			//Type Arrays
			//ARRAY OF BOOL
			IF FIND(Lynus_Standards.GVL_Communicator.arrInterfaceInfoAlVariables[byReadWriteArrayNumber,udiActiveNumberOfSymbol_ReadAds].sSymbolType,'OF BOOL') <> 0 THEN
				stADSRead_ReadAds[udiActiveNumberOfSymbol_ReadAds].sFullSymbolName := Lynus_Standards.GVL_Communicator.arrInterfaceInfoAlVariables[byReadWriteArrayNumber,udiActiveNumberOfSymbol_ReadAds].sFullSymbolName;
					stADSRead_ReadAds[udiActiveNumberOfSymbol_ReadAds].arrValue := arrValueDefault_ReadAds;	
						IF Lynus_Standards.GVL_Communicator.arrInterfaceInfoAlVariables[byReadWriteArrayNumber,udiActiveNumberOfSymbol_ReadAds].uiSizeArray <= Lynus_Standards.Constants_Communicator.bySizeOfValueArray THEN  
							FOR uiLPWriteValueByArray_ReadAds := 1 TO Lynus_Standards.GVL_Communicator.arrInterfaceInfoAlVariables[byReadWriteArrayNumber,udiActiveNumberOfSymbol_ReadAds].uiSizeArray BY 1 DO 	
								stADSRead_ReadAds[udiActiveNumberOfSymbol_ReadAds].arrValue[uiLPWriteValueByArray_ReadAds] := BYTE_TO_STRING(arrValueAfterRead_ReadAds[uiLPWriteValueByArray_ReadAds]);
							END_FOR 
						END_IF
			END_IF 
				//ARRAY OF BYTE
				IF FIND(Lynus_Standards.GVL_Communicator.arrInterfaceInfoAlVariables[byReadWriteArrayNumber,udiActiveNumberOfSymbol_ReadAds].sSymbolType,'OF BYTE') <> 0 THEN
					stADSRead_ReadAds[udiActiveNumberOfSymbol_ReadAds].sFullSymbolName := Lynus_Standards.GVL_Communicator.arrInterfaceInfoAlVariables[byReadWriteArrayNumber,udiActiveNumberOfSymbol_ReadAds].sFullSymbolName;
						stADSRead_ReadAds[udiActiveNumberOfSymbol_ReadAds].arrValue := arrValueDefault_ReadAds;	
							IF Lynus_Standards.GVL_Communicator.arrInterfaceInfoAlVariables[byReadWriteArrayNumber,udiActiveNumberOfSymbol_ReadAds].uiSizeArray <= Lynus_Standards.Constants_Communicator.bySizeOfValueArray THEN  
								FOR uiLPWriteValueByArray_ReadAds := 1 TO Lynus_Standards.GVL_Communicator.arrInterfaceInfoAlVariables[byReadWriteArrayNumber,udiActiveNumberOfSymbol_ReadAds].uiSizeArray BY 1 DO 	
									stADSRead_ReadAds[udiActiveNumberOfSymbol_ReadAds].arrValue[uiLPWriteValueByArray_ReadAds] := BYTE_TO_STRING(arrValueAfterRead_ReadAds[uiLPWriteValueByArray_ReadAds]);
								END_FOR 
							END_IF
				END_IF
			//ARRAY OF WORD
			IF FIND(Lynus_Standards.GVL_Communicator.arrInterfaceInfoAlVariables[byReadWriteArrayNumber,udiActiveNumberOfSymbol_ReadAds].sSymbolType,'OF WORD') <> 0 THEN
				stADSRead_ReadAds[udiActiveNumberOfSymbol_ReadAds].sFullSymbolName := Lynus_Standards.GVL_Communicator.arrInterfaceInfoAlVariables[byReadWriteArrayNumber,udiActiveNumberOfSymbol_ReadAds].sFullSymbolName;
					stADSRead_ReadAds[udiActiveNumberOfSymbol_ReadAds].arrValue := arrValueDefault_ReadAds;	
						IF Lynus_Standards.GVL_Communicator.arrInterfaceInfoAlVariables[byReadWriteArrayNumber,udiActiveNumberOfSymbol_ReadAds].uiSizeArray <= Lynus_Standards.Constants_Communicator.bySizeOfValueArray THEN  
							FOR uiLPWriteValueByArray_ReadAds := 1 TO Lynus_Standards.GVL_Communicator.arrInterfaceInfoAlVariables[byReadWriteArrayNumber,udiActiveNumberOfSymbol_ReadAds].uiSizeArray BY 1 DO
								arrCounterWriteValueInArray_ReadAds[1] := LIMIT(1,arrCounterWriteValueInArray_ReadAds[1],1600); arrCounterWriteValueInArray_ReadAds[2] := LIMIT(2,arrCounterWriteValueInArray_ReadAds[2],1600);
									stADSRead_ReadAds[udiActiveNumberOfSymbol_ReadAds].arrValue[uiLPWriteValueByArray_ReadAds] := WORD_TO_STRING(SHL(BYTE_TO_WORD(arrValueAfterRead_ReadAds[arrCounterWriteValueInArray_ReadAds[2]]),8) + BYTE_TO_WORD(arrValueAfterRead_ReadAds[arrCounterWriteValueInArray_ReadAds[1]]));;
								arrCounterWriteValueInArray_ReadAds[1] := arrCounterWriteValueInArray_ReadAds[1] + 2; arrCounterWriteValueInArray_ReadAds[2] := arrCounterWriteValueInArray_ReadAds[2] + 2;
							END_FOR 
						END_IF
			END_IF
				//ARRAY OF DWORD	
				IF FIND(Lynus_Standards.GVL_Communicator.arrInterfaceInfoAlVariables[byReadWriteArrayNumber,udiActiveNumberOfSymbol_ReadAds].sSymbolType,'OF DWORD') <> 0 THEN
					stADSRead_ReadAds[udiActiveNumberOfSymbol_ReadAds].sFullSymbolName := Lynus_Standards.GVL_Communicator.arrInterfaceInfoAlVariables[byReadWriteArrayNumber,udiActiveNumberOfSymbol_ReadAds].sFullSymbolName;
						stADSRead_ReadAds[udiActiveNumberOfSymbol_ReadAds].arrValue := arrValueDefault_ReadAds;	
							IF Lynus_Standards.GVL_Communicator.arrInterfaceInfoAlVariables[byReadWriteArrayNumber,udiActiveNumberOfSymbol_ReadAds].uiSizeArray <= Lynus_Standards.Constants_Communicator.bySizeOfValueArray THEN  
								FOR uiLPWriteValueByArray_ReadAds := 1 TO Lynus_Standards.GVL_Communicator.arrInterfaceInfoAlVariables[byReadWriteArrayNumber,udiActiveNumberOfSymbol_ReadAds].uiSizeArray BY 1 DO
									arrCounterWriteValueInArray_ReadAds[1] := LIMIT(1,arrCounterWriteValueInArray_ReadAds[1],1600); arrCounterWriteValueInArray_ReadAds[2] := LIMIT(2,arrCounterWriteValueInArray_ReadAds[2],1600);
										arrCounterWriteValueInArray_ReadAds[3] := LIMIT(3,arrCounterWriteValueInArray_ReadAds[3],1600); arrCounterWriteValueInArray_ReadAds[4] := LIMIT(4,arrCounterWriteValueInArray_ReadAds[4],1600);
											stADSRead_ReadAds[udiActiveNumberOfSymbol_ReadAds].arrValue[uiLPWriteValueByArray_ReadAds] := DWORD_TO_STRING(SHL(BYTE_TO_DWORD(arrValueAfterRead_ReadAds[arrCounterWriteValueInArray_ReadAds[4]]),24) + SHL(BYTE_TO_DWORD(arrValueAfterRead_ReadAds[arrCounterWriteValueInArray_ReadAds[3]]),16) + SHL(BYTE_TO_DWORD(arrValueAfterRead_ReadAds[arrCounterWriteValueInArray_ReadAds[2]]),8) + BYTE_TO_DWORD(arrValueAfterRead_ReadAds[arrCounterWriteValueInArray_ReadAds[1]]));
									arrCounterWriteValueInArray_ReadAds[1] := arrCounterWriteValueInArray_ReadAds[1] + 4; arrCounterWriteValueInArray_ReadAds[2] := arrCounterWriteValueInArray_ReadAds[2] + 4;
										arrCounterWriteValueInArray_ReadAds[3] := arrCounterWriteValueInArray_ReadAds[3] + 4; arrCounterWriteValueInArray_ReadAds[4] := arrCounterWriteValueInArray_ReadAds[4] + 4;
								END_FOR 
							END_IF
				END_IF
			//ARRAY OF SINT
			IF FIND(Lynus_Standards.GVL_Communicator.arrInterfaceInfoAlVariables[byReadWriteArrayNumber,udiActiveNumberOfSymbol_ReadAds].sSymbolType,'OF SINT') <> 0 THEN
				stADSRead_ReadAds[udiActiveNumberOfSymbol_ReadAds].sFullSymbolName := Lynus_Standards.GVL_Communicator.arrInterfaceInfoAlVariables[byReadWriteArrayNumber,udiActiveNumberOfSymbol_ReadAds].sFullSymbolName;
					stADSRead_ReadAds[udiActiveNumberOfSymbol_ReadAds].arrValue := arrValueDefault_ReadAds;	
						IF Lynus_Standards.GVL_Communicator.arrInterfaceInfoAlVariables[byReadWriteArrayNumber,udiActiveNumberOfSymbol_ReadAds].uiSizeArray <= Lynus_Standards.Constants_Communicator.bySizeOfValueArray THEN  
							FOR uiLPWriteValueByArray_ReadAds := 1 TO Lynus_Standards.GVL_Communicator.arrInterfaceInfoAlVariables[byReadWriteArrayNumber,udiActiveNumberOfSymbol_ReadAds].uiSizeArray BY 1 DO 	
								stADSRead_ReadAds[udiActiveNumberOfSymbol_ReadAds].arrValue[uiLPWriteValueByArray_ReadAds] := SINT_TO_STRING(BYTE_TO_SINT(arrValueAfterRead_ReadAds[uiLPWriteValueByArray_ReadAds]));
							END_FOR 
						END_IF
			END_IF
				//ARRAY OF USINT
				IF FIND(Lynus_Standards.GVL_Communicator.arrInterfaceInfoAlVariables[byReadWriteArrayNumber,udiActiveNumberOfSymbol_ReadAds].sSymbolType,'OF USINT') <> 0 THEN
					stADSRead_ReadAds[udiActiveNumberOfSymbol_ReadAds].sFullSymbolName := Lynus_Standards.GVL_Communicator.arrInterfaceInfoAlVariables[byReadWriteArrayNumber,udiActiveNumberOfSymbol_ReadAds].sFullSymbolName;
						stADSRead_ReadAds[udiActiveNumberOfSymbol_ReadAds].arrValue := arrValueDefault_ReadAds;	
							IF Lynus_Standards.GVL_Communicator.arrInterfaceInfoAlVariables[byReadWriteArrayNumber,udiActiveNumberOfSymbol_ReadAds].uiSizeArray <= Lynus_Standards.Constants_Communicator.bySizeOfValueArray THEN  
								FOR uiLPWriteValueByArray_ReadAds := 1 TO Lynus_Standards.GVL_Communicator.arrInterfaceInfoAlVariables[byReadWriteArrayNumber,udiActiveNumberOfSymbol_ReadAds].uiSizeArray BY 1 DO 	
									stADSRead_ReadAds[udiActiveNumberOfSymbol_ReadAds].arrValue[uiLPWriteValueByArray_ReadAds] := USINT_TO_STRING(BYTE_TO_USINT(arrValueAfterRead_ReadAds[uiLPWriteValueByArray_ReadAds]));
								END_FOR 
							END_IF
				END_IF
			//ARRAY OF INT
			IF FIND(Lynus_Standards.GVL_Communicator.arrInterfaceInfoAlVariables[byReadWriteArrayNumber,udiActiveNumberOfSymbol_ReadAds].sSymbolType,'OF INT') <> 0 THEN
				stADSRead_ReadAds[udiActiveNumberOfSymbol_ReadAds].sFullSymbolName := Lynus_Standards.GVL_Communicator.arrInterfaceInfoAlVariables[byReadWriteArrayNumber,udiActiveNumberOfSymbol_ReadAds].sFullSymbolName;
					stADSRead_ReadAds[udiActiveNumberOfSymbol_ReadAds].arrValue := arrValueDefault_ReadAds;	
						IF Lynus_Standards.GVL_Communicator.arrInterfaceInfoAlVariables[byReadWriteArrayNumber,udiActiveNumberOfSymbol_ReadAds].uiSizeArray <= Lynus_Standards.Constants_Communicator.bySizeOfValueArray THEN  
							FOR uiLPWriteValueByArray_ReadAds := 1 TO Lynus_Standards.GVL_Communicator.arrInterfaceInfoAlVariables[byReadWriteArrayNumber,udiActiveNumberOfSymbol_ReadAds].uiSizeArray BY 1 DO
								arrCounterWriteValueInArray_ReadAds[1] := LIMIT(1,arrCounterWriteValueInArray_ReadAds[1],1600); arrCounterWriteValueInArray_ReadAds[2] := LIMIT(2,arrCounterWriteValueInArray_ReadAds[2],1600);
									stADSRead_ReadAds[udiActiveNumberOfSymbol_ReadAds].arrValue[uiLPWriteValueByArray_ReadAds] := INT_TO_STRING(SHL(BYTE_TO_INT(arrValueAfterRead_ReadAds[arrCounterWriteValueInArray_ReadAds[2]]),8) + BYTE_TO_INT(arrValueAfterRead_ReadAds[arrCounterWriteValueInArray_ReadAds[1]]));;
								arrCounterWriteValueInArray_ReadAds[1] := arrCounterWriteValueInArray_ReadAds[1] + 2; arrCounterWriteValueInArray_ReadAds[2] := arrCounterWriteValueInArray_ReadAds[2] + 2;
							END_FOR 
						END_IF
			END_IF
				//ARRAY OF UINT
				IF FIND(Lynus_Standards.GVL_Communicator.arrInterfaceInfoAlVariables[byReadWriteArrayNumber,udiActiveNumberOfSymbol_ReadAds].sSymbolType,'OF UINT') <> 0 THEN
					stADSRead_ReadAds[udiActiveNumberOfSymbol_ReadAds].sFullSymbolName := Lynus_Standards.GVL_Communicator.arrInterfaceInfoAlVariables[byReadWriteArrayNumber,udiActiveNumberOfSymbol_ReadAds].sFullSymbolName;
						stADSRead_ReadAds[udiActiveNumberOfSymbol_ReadAds].arrValue := arrValueDefault_ReadAds;	
							IF Lynus_Standards.GVL_Communicator.arrInterfaceInfoAlVariables[byReadWriteArrayNumber,udiActiveNumberOfSymbol_ReadAds].uiSizeArray <= Lynus_Standards.Constants_Communicator.bySizeOfValueArray THEN  
								FOR uiLPWriteValueByArray_ReadAds := 1 TO Lynus_Standards.GVL_Communicator.arrInterfaceInfoAlVariables[byReadWriteArrayNumber,udiActiveNumberOfSymbol_ReadAds].uiSizeArray BY 1 DO
									arrCounterWriteValueInArray_ReadAds[1] := LIMIT(1,arrCounterWriteValueInArray_ReadAds[1],1600); arrCounterWriteValueInArray_ReadAds[2] := LIMIT(2,arrCounterWriteValueInArray_ReadAds[2],1600);
										stADSRead_ReadAds[udiActiveNumberOfSymbol_ReadAds].arrValue[uiLPWriteValueByArray_ReadAds] := UINT_TO_STRING(SHL(BYTE_TO_UINT(arrValueAfterRead_ReadAds[arrCounterWriteValueInArray_ReadAds[2]]),8) + BYTE_TO_UINT(arrValueAfterRead_ReadAds[arrCounterWriteValueInArray_ReadAds[1]]));;
									arrCounterWriteValueInArray_ReadAds[1] := arrCounterWriteValueInArray_ReadAds[1] + 2; arrCounterWriteValueInArray_ReadAds[2] := arrCounterWriteValueInArray_ReadAds[2] + 2;
								END_FOR 
							END_IF
				END_IF
			//ARRAY OF DINT	
			IF FIND(Lynus_Standards.GVL_Communicator.arrInterfaceInfoAlVariables[byReadWriteArrayNumber,udiActiveNumberOfSymbol_ReadAds].sSymbolType,'OF DINT') <> 0 THEN
				stADSRead_ReadAds[udiActiveNumberOfSymbol_ReadAds].sFullSymbolName := Lynus_Standards.GVL_Communicator.arrInterfaceInfoAlVariables[byReadWriteArrayNumber,udiActiveNumberOfSymbol_ReadAds].sFullSymbolName;
					stADSRead_ReadAds[udiActiveNumberOfSymbol_ReadAds].arrValue := arrValueDefault_ReadAds;	
						IF Lynus_Standards.GVL_Communicator.arrInterfaceInfoAlVariables[byReadWriteArrayNumber,udiActiveNumberOfSymbol_ReadAds].uiSizeArray <= Lynus_Standards.Constants_Communicator.bySizeOfValueArray THEN  
							FOR uiLPWriteValueByArray_ReadAds := 1 TO Lynus_Standards.GVL_Communicator.arrInterfaceInfoAlVariables[byReadWriteArrayNumber,udiActiveNumberOfSymbol_ReadAds].uiSizeArray BY 1 DO
								arrCounterWriteValueInArray_ReadAds[1] := LIMIT(1,arrCounterWriteValueInArray_ReadAds[1],1600); arrCounterWriteValueInArray_ReadAds[2] := LIMIT(2,arrCounterWriteValueInArray_ReadAds[2],1600);
									arrCounterWriteValueInArray_ReadAds[3] := LIMIT(3,arrCounterWriteValueInArray_ReadAds[3],1600); arrCounterWriteValueInArray_ReadAds[4] := LIMIT(4,arrCounterWriteValueInArray_ReadAds[4],1600);
										stADSRead_ReadAds[udiActiveNumberOfSymbol_ReadAds].arrValue[uiLPWriteValueByArray_ReadAds] := DINT_TO_STRING(SHL(BYTE_TO_DINT(arrValueAfterRead_ReadAds[arrCounterWriteValueInArray_ReadAds[4]]),24) + SHL(BYTE_TO_DINT(arrValueAfterRead_ReadAds[arrCounterWriteValueInArray_ReadAds[3]]),16) + SHL(BYTE_TO_DINT(arrValueAfterRead_ReadAds[arrCounterWriteValueInArray_ReadAds[2]]),8) + BYTE_TO_DINT(arrValueAfterRead_ReadAds[arrCounterWriteValueInArray_ReadAds[1]]));
								arrCounterWriteValueInArray_ReadAds[1] := arrCounterWriteValueInArray_ReadAds[1] + 4; arrCounterWriteValueInArray_ReadAds[2] := arrCounterWriteValueInArray_ReadAds[2] + 4;
									arrCounterWriteValueInArray_ReadAds[3] := arrCounterWriteValueInArray_ReadAds[3] + 4; arrCounterWriteValueInArray_ReadAds[4] := arrCounterWriteValueInArray_ReadAds[4] + 4;
							END_FOR 
						END_IF
			END_IF
				//ARRAY OF UDINT	
				IF FIND(Lynus_Standards.GVL_Communicator.arrInterfaceInfoAlVariables[byReadWriteArrayNumber,udiActiveNumberOfSymbol_ReadAds].sSymbolType,'OF UDINT') <> 0 THEN
					stADSRead_ReadAds[udiActiveNumberOfSymbol_ReadAds].sFullSymbolName := Lynus_Standards.GVL_Communicator.arrInterfaceInfoAlVariables[byReadWriteArrayNumber,udiActiveNumberOfSymbol_ReadAds].sFullSymbolName;
						stADSRead_ReadAds[udiActiveNumberOfSymbol_ReadAds].arrValue := arrValueDefault_ReadAds;	
							IF Lynus_Standards.GVL_Communicator.arrInterfaceInfoAlVariables[byReadWriteArrayNumber,udiActiveNumberOfSymbol_ReadAds].uiSizeArray <= Lynus_Standards.Constants_Communicator.bySizeOfValueArray THEN  
								FOR uiLPWriteValueByArray_ReadAds := 1 TO Lynus_Standards.GVL_Communicator.arrInterfaceInfoAlVariables[byReadWriteArrayNumber,udiActiveNumberOfSymbol_ReadAds].uiSizeArray BY 1 DO
									arrCounterWriteValueInArray_ReadAds[1] := LIMIT(1,arrCounterWriteValueInArray_ReadAds[1],1600); arrCounterWriteValueInArray_ReadAds[2] := LIMIT(2,arrCounterWriteValueInArray_ReadAds[2],1600);
										arrCounterWriteValueInArray_ReadAds[3] := LIMIT(3,arrCounterWriteValueInArray_ReadAds[3],1600); arrCounterWriteValueInArray_ReadAds[4] := LIMIT(4,arrCounterWriteValueInArray_ReadAds[4],1600);
											stADSRead_ReadAds[udiActiveNumberOfSymbol_ReadAds].arrValue[uiLPWriteValueByArray_ReadAds] := UDINT_TO_STRING(SHL(BYTE_TO_UDINT(arrValueAfterRead_ReadAds[arrCounterWriteValueInArray_ReadAds[4]]),24) + SHL(BYTE_TO_UDINT(arrValueAfterRead_ReadAds[arrCounterWriteValueInArray_ReadAds[3]]),16) + SHL(BYTE_TO_UDINT(arrValueAfterRead_ReadAds[arrCounterWriteValueInArray_ReadAds[2]]),8) + BYTE_TO_UDINT(arrValueAfterRead_ReadAds[arrCounterWriteValueInArray_ReadAds[1]]));
									arrCounterWriteValueInArray_ReadAds[1] := arrCounterWriteValueInArray_ReadAds[1] + 4; arrCounterWriteValueInArray_ReadAds[2] := arrCounterWriteValueInArray_ReadAds[2] + 4;
										arrCounterWriteValueInArray_ReadAds[3] := arrCounterWriteValueInArray_ReadAds[3] + 4; arrCounterWriteValueInArray_ReadAds[4] := arrCounterWriteValueInArray_ReadAds[4] + 4;
								END_FOR 
							END_IF
				END_IF
					//ARRAY OF LINT	
					IF FIND(Lynus_Standards.GVL_Communicator.arrInterfaceInfoAlVariables[byReadWriteArrayNumber,udiActiveNumberOfSymbol_ReadAds].sSymbolType,'OF LINT') <> 0 THEN
						stADSRead_ReadAds[udiActiveNumberOfSymbol_ReadAds].sFullSymbolName := Lynus_Standards.GVL_Communicator.arrInterfaceInfoAlVariables[byReadWriteArrayNumber,udiActiveNumberOfSymbol_ReadAds].sFullSymbolName;
							stADSRead_ReadAds[udiActiveNumberOfSymbol_ReadAds].arrValue := arrValueDefault_ReadAds;	
								IF Lynus_Standards.GVL_Communicator.arrInterfaceInfoAlVariables[byReadWriteArrayNumber,udiActiveNumberOfSymbol_ReadAds].uiSizeArray <= Lynus_Standards.Constants_Communicator.bySizeOfValueArray THEN  
									FOR uiLPWriteValueByArray_ReadAds := 1 TO Lynus_Standards.GVL_Communicator.arrInterfaceInfoAlVariables[byReadWriteArrayNumber,udiActiveNumberOfSymbol_ReadAds].uiSizeArray BY 1 DO
										arrCounterWriteValueInArray_ReadAds[1] := LIMIT(1,arrCounterWriteValueInArray_ReadAds[1],1600); arrCounterWriteValueInArray_ReadAds[2] := LIMIT(2,arrCounterWriteValueInArray_ReadAds[2],1600);
											arrCounterWriteValueInArray_ReadAds[3] := LIMIT(3,arrCounterWriteValueInArray_ReadAds[3],1600); arrCounterWriteValueInArray_ReadAds[4] := LIMIT(4,arrCounterWriteValueInArray_ReadAds[4],1600);
												arrCounterWriteValueInArray_ReadAds[5] := LIMIT(5,arrCounterWriteValueInArray_ReadAds[5],1600); arrCounterWriteValueInArray_ReadAds[6] := LIMIT(6,arrCounterWriteValueInArray_ReadAds[6],1600);
													arrCounterWriteValueInArray_ReadAds[7] := LIMIT(7,arrCounterWriteValueInArray_ReadAds[7],1600); arrCounterWriteValueInArray_ReadAds[8] := LIMIT(8,arrCounterWriteValueInArray_ReadAds[8],1600);
														stADSRead_ReadAds[udiActiveNumberOfSymbol_ReadAds].arrValue[uiLPWriteValueByArray_ReadAds] := LINT_TO_STRING(SHL(BYTE_TO_LINT(arrValueAfterRead_ReadAds[arrCounterWriteValueInArray_ReadAds[8]]),56) + SHL(BYTE_TO_LINT(arrValueAfterRead_ReadAds[arrCounterWriteValueInArray_ReadAds[7]]),48) + SHL(BYTE_TO_LINT(arrValueAfterRead_ReadAds[arrCounterWriteValueInArray_ReadAds[6]]),40) + SHL(BYTE_TO_LINT(arrValueAfterRead_ReadAds[arrCounterWriteValueInArray_ReadAds[5]]),32) +
																																							SHL(BYTE_TO_LINT(arrValueAfterRead_ReadAds[arrCounterWriteValueInArray_ReadAds[4]]),24) + SHL(BYTE_TO_LINT(arrValueAfterRead_ReadAds[arrCounterWriteValueInArray_ReadAds[3]]),16) + SHL(BYTE_TO_LINT(arrValueAfterRead_ReadAds[arrCounterWriteValueInArray_ReadAds[2]]),8) + BYTE_TO_LINT(arrValueAfterRead_ReadAds[arrCounterWriteValueInArray_ReadAds[1]]));
										arrCounterWriteValueInArray_ReadAds[1] := arrCounterWriteValueInArray_ReadAds[1] + 8; arrCounterWriteValueInArray_ReadAds[2] := arrCounterWriteValueInArray_ReadAds[2] + 8;
											arrCounterWriteValueInArray_ReadAds[3] := arrCounterWriteValueInArray_ReadAds[3] + 8; arrCounterWriteValueInArray_ReadAds[4] := arrCounterWriteValueInArray_ReadAds[4] + 8;
												arrCounterWriteValueInArray_ReadAds[5] := arrCounterWriteValueInArray_ReadAds[5] + 8; arrCounterWriteValueInArray_ReadAds[6] := arrCounterWriteValueInArray_ReadAds[6] + 8;
													arrCounterWriteValueInArray_ReadAds[7] := arrCounterWriteValueInArray_ReadAds[7] + 8; arrCounterWriteValueInArray_ReadAds[8] := arrCounterWriteValueInArray_ReadAds[8] + 8;
									END_FOR 
								END_IF
					END_IF
				//ARRAY OF ULINT	
				IF FIND(Lynus_Standards.GVL_Communicator.arrInterfaceInfoAlVariables[byReadWriteArrayNumber,udiActiveNumberOfSymbol_ReadAds].sSymbolType,'OF ULINT') <> 0 THEN
					stADSRead_ReadAds[udiActiveNumberOfSymbol_ReadAds].sFullSymbolName := Lynus_Standards.GVL_Communicator.arrInterfaceInfoAlVariables[byReadWriteArrayNumber,udiActiveNumberOfSymbol_ReadAds].sFullSymbolName;
						stADSRead_ReadAds[udiActiveNumberOfSymbol_ReadAds].arrValue := arrValueDefault_ReadAds;	
							IF Lynus_Standards.GVL_Communicator.arrInterfaceInfoAlVariables[byReadWriteArrayNumber,udiActiveNumberOfSymbol_ReadAds].uiSizeArray <= Lynus_Standards.Constants_Communicator.bySizeOfValueArray THEN  
								FOR uiLPWriteValueByArray_ReadAds := 1 TO Lynus_Standards.GVL_Communicator.arrInterfaceInfoAlVariables[byReadWriteArrayNumber,udiActiveNumberOfSymbol_ReadAds].uiSizeArray BY 1 DO
									arrCounterWriteValueInArray_ReadAds[1] := LIMIT(1,arrCounterWriteValueInArray_ReadAds[1],1600); arrCounterWriteValueInArray_ReadAds[2] := LIMIT(2,arrCounterWriteValueInArray_ReadAds[2],1600);
										arrCounterWriteValueInArray_ReadAds[3] := LIMIT(3,arrCounterWriteValueInArray_ReadAds[3],1600); arrCounterWriteValueInArray_ReadAds[4] := LIMIT(4,arrCounterWriteValueInArray_ReadAds[4],1600);
											arrCounterWriteValueInArray_ReadAds[5] := LIMIT(5,arrCounterWriteValueInArray_ReadAds[5],1600); arrCounterWriteValueInArray_ReadAds[6] := LIMIT(6,arrCounterWriteValueInArray_ReadAds[6],1600);
												arrCounterWriteValueInArray_ReadAds[7] := LIMIT(7,arrCounterWriteValueInArray_ReadAds[7],1600); arrCounterWriteValueInArray_ReadAds[8] := LIMIT(8,arrCounterWriteValueInArray_ReadAds[8],1600);
													stADSRead_ReadAds[udiActiveNumberOfSymbol_ReadAds].arrValue[uiLPWriteValueByArray_ReadAds] := ULINT_TO_STRING(SHL(BYTE_TO_ULINT(arrValueAfterRead_ReadAds[arrCounterWriteValueInArray_ReadAds[8]]),56) + SHL(BYTE_TO_ULINT(arrValueAfterRead_ReadAds[arrCounterWriteValueInArray_ReadAds[7]]),48) + SHL(BYTE_TO_ULINT(arrValueAfterRead_ReadAds[arrCounterWriteValueInArray_ReadAds[6]]),40) + SHL(BYTE_TO_ULINT(arrValueAfterRead_ReadAds[arrCounterWriteValueInArray_ReadAds[5]]),32) +
																																						SHL(BYTE_TO_ULINT(arrValueAfterRead_ReadAds[arrCounterWriteValueInArray_ReadAds[4]]),24) + SHL(BYTE_TO_ULINT(arrValueAfterRead_ReadAds[arrCounterWriteValueInArray_ReadAds[3]]),16) + SHL(BYTE_TO_ULINT(arrValueAfterRead_ReadAds[arrCounterWriteValueInArray_ReadAds[2]]),8) + BYTE_TO_ULINT(arrValueAfterRead_ReadAds[arrCounterWriteValueInArray_ReadAds[1]]));
									arrCounterWriteValueInArray_ReadAds[1] := arrCounterWriteValueInArray_ReadAds[1] + 8; arrCounterWriteValueInArray_ReadAds[2] := arrCounterWriteValueInArray_ReadAds[2] + 8;
										arrCounterWriteValueInArray_ReadAds[3] := arrCounterWriteValueInArray_ReadAds[3] + 8; arrCounterWriteValueInArray_ReadAds[4] := arrCounterWriteValueInArray_ReadAds[4] + 8;
											arrCounterWriteValueInArray_ReadAds[5] := arrCounterWriteValueInArray_ReadAds[5] + 8; arrCounterWriteValueInArray_ReadAds[6] := arrCounterWriteValueInArray_ReadAds[6] + 8;
												arrCounterWriteValueInArray_ReadAds[7] := arrCounterWriteValueInArray_ReadAds[7] + 8; arrCounterWriteValueInArray_ReadAds[8] := arrCounterWriteValueInArray_ReadAds[8] + 8;
								END_FOR 
							END_IF
				END_IF
					//ARRAY OF LWORD	
					IF FIND(Lynus_Standards.GVL_Communicator.arrInterfaceInfoAlVariables[byReadWriteArrayNumber,udiActiveNumberOfSymbol_ReadAds].sSymbolType,'OF LWORD') <> 0 THEN
						stADSRead_ReadAds[udiActiveNumberOfSymbol_ReadAds].sFullSymbolName := Lynus_Standards.GVL_Communicator.arrInterfaceInfoAlVariables[byReadWriteArrayNumber,udiActiveNumberOfSymbol_ReadAds].sFullSymbolName;
							stADSRead_ReadAds[udiActiveNumberOfSymbol_ReadAds].arrValue := arrValueDefault_ReadAds;	
								IF Lynus_Standards.GVL_Communicator.arrInterfaceInfoAlVariables[byReadWriteArrayNumber,udiActiveNumberOfSymbol_ReadAds].uiSizeArray <= Lynus_Standards.Constants_Communicator.bySizeOfValueArray THEN  
									FOR uiLPWriteValueByArray_ReadAds := 1 TO Lynus_Standards.GVL_Communicator.arrInterfaceInfoAlVariables[byReadWriteArrayNumber,udiActiveNumberOfSymbol_ReadAds].uiSizeArray BY 1 DO
										arrCounterWriteValueInArray_ReadAds[1] := LIMIT(1,arrCounterWriteValueInArray_ReadAds[1],1600); arrCounterWriteValueInArray_ReadAds[2] := LIMIT(2,arrCounterWriteValueInArray_ReadAds[2],1600);
											arrCounterWriteValueInArray_ReadAds[3] := LIMIT(3,arrCounterWriteValueInArray_ReadAds[3],1600); arrCounterWriteValueInArray_ReadAds[4] := LIMIT(4,arrCounterWriteValueInArray_ReadAds[4],1600);
												arrCounterWriteValueInArray_ReadAds[5] := LIMIT(5,arrCounterWriteValueInArray_ReadAds[5],1600); arrCounterWriteValueInArray_ReadAds[6] := LIMIT(6,arrCounterWriteValueInArray_ReadAds[6],1600);
													arrCounterWriteValueInArray_ReadAds[7] := LIMIT(7,arrCounterWriteValueInArray_ReadAds[7],1600); arrCounterWriteValueInArray_ReadAds[8] := LIMIT(8,arrCounterWriteValueInArray_ReadAds[8],1600);
														stADSRead_ReadAds[udiActiveNumberOfSymbol_ReadAds].arrValue[uiLPWriteValueByArray_ReadAds] := LWORD_TO_STRING(SHL(BYTE_TO_LWORD(arrValueAfterRead_ReadAds[arrCounterWriteValueInArray_ReadAds[8]]),56) + SHL(BYTE_TO_LWORD(arrValueAfterRead_ReadAds[arrCounterWriteValueInArray_ReadAds[7]]),48) + SHL(BYTE_TO_LWORD(arrValueAfterRead_ReadAds[arrCounterWriteValueInArray_ReadAds[6]]),40) + SHL(BYTE_TO_LWORD(arrValueAfterRead_ReadAds[arrCounterWriteValueInArray_ReadAds[5]]),32) +
																																							SHL(BYTE_TO_LWORD(arrValueAfterRead_ReadAds[arrCounterWriteValueInArray_ReadAds[4]]),24) + SHL(BYTE_TO_LWORD(arrValueAfterRead_ReadAds[arrCounterWriteValueInArray_ReadAds[3]]),16) + SHL(BYTE_TO_LWORD(arrValueAfterRead_ReadAds[arrCounterWriteValueInArray_ReadAds[2]]),8) + BYTE_TO_LWORD(arrValueAfterRead_ReadAds[arrCounterWriteValueInArray_ReadAds[1]]));
										arrCounterWriteValueInArray_ReadAds[1] := arrCounterWriteValueInArray_ReadAds[1] + 8; arrCounterWriteValueInArray_ReadAds[2] := arrCounterWriteValueInArray_ReadAds[2] + 8;
											arrCounterWriteValueInArray_ReadAds[3] := arrCounterWriteValueInArray_ReadAds[3] + 8; arrCounterWriteValueInArray_ReadAds[4] := arrCounterWriteValueInArray_ReadAds[4] + 8;
												arrCounterWriteValueInArray_ReadAds[5] := arrCounterWriteValueInArray_ReadAds[5] + 8; arrCounterWriteValueInArray_ReadAds[6] := arrCounterWriteValueInArray_ReadAds[6] + 8;
													arrCounterWriteValueInArray_ReadAds[7] := arrCounterWriteValueInArray_ReadAds[7] + 8; arrCounterWriteValueInArray_ReadAds[8] := arrCounterWriteValueInArray_ReadAds[8] + 8;
									END_FOR 
								END_IF
					END_IF
				//ARRAY OF REAL
				IF FIND(Lynus_Standards.GVL_Communicator.arrInterfaceInfoAlVariables[byReadWriteArrayNumber,udiActiveNumberOfSymbol_ReadAds].sSymbolType,'OF REAL') <> 0 THEN
					stADSRead_ReadAds[udiActiveNumberOfSymbol_ReadAds].sFullSymbolName := Lynus_Standards.GVL_Communicator.arrInterfaceInfoAlVariables[byReadWriteArrayNumber,udiActiveNumberOfSymbol_ReadAds].sFullSymbolName;
						stADSRead_ReadAds[udiActiveNumberOfSymbol_ReadAds].arrValue := arrValueDefault_ReadAds;	
							IF Lynus_Standards.GVL_Communicator.arrInterfaceInfoAlVariables[byReadWriteArrayNumber,udiActiveNumberOfSymbol_ReadAds].uiSizeArray <= Lynus_Standards.Constants_Communicator.bySizeOfValueArray THEN  
								FOR uiLPWriteValueByArray_ReadAds := 1 TO Lynus_Standards.GVL_Communicator.arrInterfaceInfoAlVariables[byReadWriteArrayNumber,udiActiveNumberOfSymbol_ReadAds].uiSizeArray BY 1 DO
									arrCounterWriteValueInArray_ReadAds[1] := LIMIT(1,arrCounterWriteValueInArray_ReadAds[1],1600); arrCounterWriteValueInArray_ReadAds[2] := LIMIT(2,arrCounterWriteValueInArray_ReadAds[2],1600);
										arrCounterWriteValueInArray_ReadAds[3] := LIMIT(3,arrCounterWriteValueInArray_ReadAds[3],1600); arrCounterWriteValueInArray_ReadAds[4] := LIMIT(4,arrCounterWriteValueInArray_ReadAds[4],1600);
											unConvertDWORD_TO_REAL_ReadAds.dwRawValue := DINT_TO_DWORD(DWORD_TO_DINT(SHL(BYTE_TO_DWORD(arrValueAfterRead_ReadAds[arrCounterWriteValueInArray_ReadAds[4]]),24) + SHL(BYTE_TO_DWORD(arrValueAfterRead_ReadAds[arrCounterWriteValueInArray_ReadAds[3]]),16) + SHL(BYTE_TO_DWORD(arrValueAfterRead_ReadAds[arrCounterWriteValueInArray_ReadAds[2]]),8) + BYTE_TO_DWORD(arrValueAfterRead_ReadAds[arrCounterWriteValueInArray_ReadAds[1]])));
									arrCounterWriteValueInArray_ReadAds[1] := arrCounterWriteValueInArray_ReadAds[1] + 4; arrCounterWriteValueInArray_ReadAds[2] := arrCounterWriteValueInArray_ReadAds[2] + 4;
										arrCounterWriteValueInArray_ReadAds[3] := arrCounterWriteValueInArray_ReadAds[3] + 4; arrCounterWriteValueInArray_ReadAds[4] := arrCounterWriteValueInArray_ReadAds[4] + 4;					
											IF IsFinite(F_REAL(unConvertDWORD_TO_REAL_ReadAds.rValueFloat)) THEN 
												IF LEN(REAL_TO_STRING(unConvertDWORD_TO_REAL_ReadAds.rValueFloat)) <= 30 THEN 
													IF FIND(REAL_TO_STRING(unConvertDWORD_TO_REAL_ReadAds.rValueFloat),'e') = 0 AND FIND(REAL_TO_STRING(unConvertDWORD_TO_REAL_ReadAds.rValueFloat),'E') = 0 THEN 
														sStringFloat_ReadAds := REAL_TO_STRING(unConvertDWORD_TO_REAL_ReadAds.rValueFloat);
															iFindPointFloat_ReadAds := FIND(sStringFloat_ReadAds,'.');
																sStringFloat_ReadAds := DELETE(sStringFloat_ReadAds,iFindPointFloat_ReadAds,1);
																	iPrecision_ReadAds := LEN(sStringFloat_ReadAds);
																		iPrecision_ReadAds := LIMIT(0,iPrecision_ReadAds,8);
														IF LEN(LREAL_TO_FMTSTR(REAL_TO_LREAL(unConvertDWORD_TO_REAL_ReadAds.rValueFloat),iPrecision_ReadAds,TRUE)) <= 30 THEN	 			
															//Check if the output from Function LREAL_TO_FMTSTR is ok 
															IF LREAL_TO_FMTSTR(REAL_TO_LREAL(unConvertDWORD_TO_REAL_ReadAds.rValueFloat),iPrecision_ReadAds,TRUE) <> '#INF' AND LREAL_TO_FMTSTR(REAL_TO_LREAL(unConvertDWORD_TO_REAL_ReadAds.rValueFloat),iPrecision_ReadAds,TRUE) <> '-#INF' AND
																LREAL_TO_FMTSTR(REAL_TO_LREAL(unConvertDWORD_TO_REAL_ReadAds.rValueFloat),iPrecision_ReadAds,TRUE) <> '#QNAN' AND LREAL_TO_FMTSTR(REAL_TO_LREAL(unConvertDWORD_TO_REAL_ReadAds.rValueFloat),iPrecision_ReadAds,TRUE) <> '-#QNAN' AND
																	LREAL_TO_FMTSTR(REAL_TO_LREAL(unConvertDWORD_TO_REAL_ReadAds.rValueFloat),iPrecision_ReadAds,TRUE) <> '#OVF' AND LREAL_TO_FMTSTR(REAL_TO_LREAL(unConvertDWORD_TO_REAL_ReadAds.rValueFloat),iPrecision_ReadAds,TRUE) <> '-#OVF' THEN	   	 			
																		stADSRead_ReadAds[udiActiveNumberOfSymbol_ReadAds].arrValue[uiLPWriteValueByArray_ReadAds] := LREAL_TO_FMTSTR(REAL_TO_LREAL(unConvertDWORD_TO_REAL_ReadAds.rValueFloat),iPrecision_ReadAds,TRUE);
															ELSE
																iState_ReadAds := 200;
																	uiInternError_ReadAds := 1;
															END_IF
														ELSE
															//Check if the output from Function LREAL_TO_FMTSTR is ok 
															IF MID(LREAL_TO_FMTSTR(REAL_TO_LREAL(unConvertDWORD_TO_REAL_ReadAds.rValueFloat),iPrecision_ReadAds,TRUE),30,1) <> '#INF' AND MID(LREAL_TO_FMTSTR(REAL_TO_LREAL(unConvertDWORD_TO_REAL_ReadAds.rValueFloat),iPrecision_ReadAds,TRUE),30,1) <> '-#INF' AND
																MID(LREAL_TO_FMTSTR(REAL_TO_LREAL(unConvertDWORD_TO_REAL_ReadAds.rValueFloat),iPrecision_ReadAds,TRUE),30,1) <> '#QNAN' AND MID(LREAL_TO_FMTSTR(REAL_TO_LREAL(unConvertDWORD_TO_REAL_ReadAds.rValueFloat),iPrecision_ReadAds,TRUE),30,1) <> '-#QNAN' AND
																	MID(LREAL_TO_FMTSTR(REAL_TO_LREAL(unConvertDWORD_TO_REAL_ReadAds.rValueFloat),iPrecision_ReadAds,TRUE),30,1) <> '#OVF' AND MID(LREAL_TO_FMTSTR(REAL_TO_LREAL(unConvertDWORD_TO_REAL_ReadAds.rValueFloat),iPrecision_ReadAds,TRUE),30,1) <> '-#OVF' THEN 
																		stADSRead_ReadAds[udiActiveNumberOfSymbol_ReadAds].arrValue[uiLPWriteValueByArray_ReadAds] := MID(LREAL_TO_FMTSTR(REAL_TO_LREAL(unConvertDWORD_TO_REAL_ReadAds.rValueFloat),iPrecision_ReadAds,TRUE),30,1);
															ELSE
																iState_ReadAds := 200;
																	uiInternError_ReadAds := 1;
															END_IF
														END_IF
													ELSE
														stADSRead_ReadAds[udiActiveNumberOfSymbol_ReadAds].arrValue[uiLPWriteValueByArray_ReadAds] := REAL_TO_STRING(unConvertDWORD_TO_REAL_ReadAds.rValueFloat);
													END_IF 
												ELSE
													iState_ReadAds := 200;
														uiInternError_ReadAds := 1;
												END_IF
											ELSE
												iState_ReadAds := 200;
													uiInternError_ReadAds := 1;	
											END_IF
								END_FOR 
							END_IF
				END_IF
					//ARRAY OF LREAL
					IF FIND(Lynus_Standards.GVL_Communicator.arrInterfaceInfoAlVariables[byReadWriteArrayNumber,udiActiveNumberOfSymbol_ReadAds].sSymbolType,'OF LREAL') <> 0 THEN
						stADSRead_ReadAds[udiActiveNumberOfSymbol_ReadAds].sFullSymbolName := Lynus_Standards.GVL_Communicator.arrInterfaceInfoAlVariables[byReadWriteArrayNumber,udiActiveNumberOfSymbol_ReadAds].sFullSymbolName;
							stADSRead_ReadAds[udiActiveNumberOfSymbol_ReadAds].arrValue := arrValueDefault_ReadAds;	
								IF Lynus_Standards.GVL_Communicator.arrInterfaceInfoAlVariables[byReadWriteArrayNumber,udiActiveNumberOfSymbol_ReadAds].uiSizeArray <= Lynus_Standards.Constants_Communicator.bySizeOfValueArray THEN  
									FOR uiLPWriteValueByArray_ReadAds := 1 TO Lynus_Standards.GVL_Communicator.arrInterfaceInfoAlVariables[byReadWriteArrayNumber,udiActiveNumberOfSymbol_ReadAds].uiSizeArray BY 1 DO
										arrCounterWriteValueInArray_ReadAds[1] := LIMIT(1,arrCounterWriteValueInArray_ReadAds[1],1600); arrCounterWriteValueInArray_ReadAds[2] := LIMIT(2,arrCounterWriteValueInArray_ReadAds[2],1600);
											arrCounterWriteValueInArray_ReadAds[3] := LIMIT(3,arrCounterWriteValueInArray_ReadAds[3],1600); arrCounterWriteValueInArray_ReadAds[4] := LIMIT(4,arrCounterWriteValueInArray_ReadAds[4],1600);
												arrCounterWriteValueInArray_ReadAds[5] := LIMIT(5,arrCounterWriteValueInArray_ReadAds[5],1600); arrCounterWriteValueInArray_ReadAds[6] := LIMIT(6,arrCounterWriteValueInArray_ReadAds[6],1600);
													arrCounterWriteValueInArray_ReadAds[7] := LIMIT(7,arrCounterWriteValueInArray_ReadAds[7],1600); arrCounterWriteValueInArray_ReadAds[8] := LIMIT(8,arrCounterWriteValueInArray_ReadAds[8],1600);
														unConvertULINT_TO_LREAL_ReadAds.uliRawValue := LINT_TO_ULINT(ULINT_TO_LINT(SHL(BYTE_TO_ULINT(arrValueAfterRead_ReadAds[arrCounterWriteValueInArray_ReadAds[8]]),56) + SHL(BYTE_TO_ULINT(arrValueAfterRead_ReadAds[arrCounterWriteValueInArray_ReadAds[7]]),48) + SHL(BYTE_TO_ULINT(arrValueAfterRead_ReadAds[arrCounterWriteValueInArray_ReadAds[6]]),40) + SHL(BYTE_TO_ULINT(arrValueAfterRead_ReadAds[arrCounterWriteValueInArray_ReadAds[5]]),32) +
																											SHL(BYTE_TO_ULINT(arrValueAfterRead_ReadAds[arrCounterWriteValueInArray_ReadAds[4]]),24) + SHL(BYTE_TO_ULINT(arrValueAfterRead_ReadAds[arrCounterWriteValueInArray_ReadAds[3]]),16) + SHL(BYTE_TO_ULINT(arrValueAfterRead_ReadAds[arrCounterWriteValueInArray_ReadAds[2]]),8) + BYTE_TO_ULINT(arrValueAfterRead_ReadAds[arrCounterWriteValueInArray_ReadAds[1]])));
										arrCounterWriteValueInArray_ReadAds[1] := arrCounterWriteValueInArray_ReadAds[1] + 8; arrCounterWriteValueInArray_ReadAds[2] := arrCounterWriteValueInArray_ReadAds[2] + 8;
											arrCounterWriteValueInArray_ReadAds[3] := arrCounterWriteValueInArray_ReadAds[3] + 8; arrCounterWriteValueInArray_ReadAds[4] := arrCounterWriteValueInArray_ReadAds[4] + 8;
												arrCounterWriteValueInArray_ReadAds[5] := arrCounterWriteValueInArray_ReadAds[5] + 8; arrCounterWriteValueInArray_ReadAds[6] := arrCounterWriteValueInArray_ReadAds[6] + 8;
													arrCounterWriteValueInArray_ReadAds[7] := arrCounterWriteValueInArray_ReadAds[7] + 8; arrCounterWriteValueInArray_ReadAds[8] := arrCounterWriteValueInArray_ReadAds[8] + 8;			
														IF IsFinite(F_LREAL(unConvertULINT_TO_LREAL_ReadAds.lrValueFloat)) THEN
															IF LEN(LREAL_TO_STRING(unConvertULINT_TO_LREAL_ReadAds.lrValueFloat)) <= 30 THEN 
																IF FIND(LREAL_TO_STRING(unConvertULINT_TO_LREAL_ReadAds.lrValueFloat),'e') = 0 AND FIND(LREAL_TO_STRING(unConvertULINT_TO_LREAL_ReadAds.lrValueFloat),'E') = 0 THEN 
																	sStringFloat_ReadAds := LREAL_TO_STRING(unConvertULINT_TO_LREAL_ReadAds.lrValueFloat);
																		iFindPointFloat_ReadAds := FIND(sStringFloat_ReadAds,'.');
																			sStringFloat_ReadAds := DELETE(sStringFloat_ReadAds,iFindPointFloat_ReadAds,1);
																				iPrecision_ReadAds := LEN(sStringFloat_ReadAds);
																					iPrecision_ReadAds := LIMIT(0,iPrecision_ReadAds,16);
																	IF LEN(LREAL_TO_FMTSTR(unConvertULINT_TO_LREAL_ReadAds.lrValueFloat,iPrecision_ReadAds,TRUE)) <= 30 THEN
																		//Check if the output from Function LREAL_TO_FMTSTR is ok 
																		IF LREAL_TO_FMTSTR(unConvertULINT_TO_LREAL_ReadAds.lrValueFloat,iPrecision_ReadAds,TRUE) <> '#INF' AND LREAL_TO_FMTSTR(unConvertULINT_TO_LREAL_ReadAds.lrValueFloat,iPrecision_ReadAds,TRUE) <> '-#INF' AND
																			LREAL_TO_FMTSTR(unConvertULINT_TO_LREAL_ReadAds.lrValueFloat,iPrecision_ReadAds,TRUE) <> '#QNAN' AND LREAL_TO_FMTSTR(unConvertULINT_TO_LREAL_ReadAds.lrValueFloat,iPrecision_ReadAds,TRUE) <> '-#QNAN' AND
																				LREAL_TO_FMTSTR(unConvertULINT_TO_LREAL_ReadAds.lrValueFloat,iPrecision_ReadAds,TRUE) <> '#OVF' AND LREAL_TO_FMTSTR(unConvertULINT_TO_LREAL_ReadAds.lrValueFloat,iPrecision_ReadAds,TRUE) <> '-#OVF' THEN
																					stADSRead_ReadAds[udiActiveNumberOfSymbol_ReadAds].arrValue[uiLPWriteValueByArray_ReadAds] := LREAL_TO_FMTSTR(unConvertULINT_TO_LREAL_ReadAds.lrValueFloat,iPrecision_ReadAds,TRUE); 
																		ELSE
																			iState_ReadAds := 200;
																				uiInternError_ReadAds := 1;
																		END_IF
																	ELSE
																		//Check if the output from Function LREAL_TO_FMTSTR is ok 
																		IF MID(LREAL_TO_FMTSTR(unConvertULINT_TO_LREAL_ReadAds.lrValueFloat,iPrecision_ReadAds,TRUE),30,1) <> '#INF' AND MID(LREAL_TO_FMTSTR(unConvertULINT_TO_LREAL_ReadAds.lrValueFloat,iPrecision_ReadAds,TRUE),30,1) <> '-#INF' AND
																			MID(LREAL_TO_FMTSTR(unConvertULINT_TO_LREAL_ReadAds.lrValueFloat,iPrecision_ReadAds,TRUE),30,1) <> '#QNAN' AND MID(LREAL_TO_FMTSTR(unConvertULINT_TO_LREAL_ReadAds.lrValueFloat,iPrecision_ReadAds,TRUE),30,1) <> '-#QNAN' AND
																				MID(LREAL_TO_FMTSTR(unConvertULINT_TO_LREAL_ReadAds.lrValueFloat,iPrecision_ReadAds,TRUE),30,1) <> '#OVF' AND MID(LREAL_TO_FMTSTR(unConvertULINT_TO_LREAL_ReadAds.lrValueFloat,iPrecision_ReadAds,TRUE),30,1) <> '-#OVF' THEN
																					stADSRead_ReadAds[udiActiveNumberOfSymbol_ReadAds].arrValue[uiLPWriteValueByArray_ReadAds] := MID(LREAL_TO_FMTSTR(unConvertULINT_TO_LREAL_ReadAds.lrValueFloat,iPrecision_ReadAds,TRUE),30,1);
																		ELSE
																			iState_ReadAds := 200;
																				uiInternError_ReadAds := 1;
																		END_IF 
																	END_IF
																ELSE
																	stADSRead_ReadAds[udiActiveNumberOfSymbol_ReadAds].arrValue[uiLPWriteValueByArray_ReadAds] := LREAL_TO_STRING(unConvertULINT_TO_LREAL_ReadAds.lrValueFloat);
																END_IF
															ELSE
																iState_ReadAds := 200;
																	uiInternError_ReadAds := 1;
															END_IF
														ELSE
															iState_ReadAds := 200;
																uiInternError_ReadAds := 1;
														END_IF
									END_FOR 
								END_IF
					END_IF
				//ARRAY OF STRING(30)
				IF FIND(Lynus_Standards.GVL_Communicator.arrInterfaceInfoAlVariables[byReadWriteArrayNumber,udiActiveNumberOfSymbol_ReadAds].sSymbolType,'OF STRING(30)') <> 0 THEN
					stADSRead_ReadAds[udiActiveNumberOfSymbol_ReadAds].sFullSymbolName := Lynus_Standards.GVL_Communicator.arrInterfaceInfoAlVariables[byReadWriteArrayNumber,udiActiveNumberOfSymbol_ReadAds].sFullSymbolName;
						stADSRead_ReadAds[udiActiveNumberOfSymbol_ReadAds].arrValue := arrValueDefault_ReadAds;	
							IF Lynus_Standards.GVL_Communicator.arrInterfaceInfoAlVariables[byReadWriteArrayNumber,udiActiveNumberOfSymbol_ReadAds].uiSizeArray <= Lynus_Standards.Constants_Communicator.bySizeOfValueArray THEN
								FOR uiLPWriteValueByArray_ReadAds := 1 TO Lynus_Standards.Constants_Communicator.bySizeOfValueArray BY 1 DO 
									FOR byLPCheckCharactersAfterReadOut_ReadAds := 1 TO 31 BY 1 DO
										uiCounterArrayOfString_ReadAds := uiCounterArrayOfString_ReadAds + 1;
											uiCounterArrayOfString_ReadAds := LIMIT(1,uiCounterArrayOfString_ReadAds,1600);	
												stADSRead_ReadAds[udiActiveNumberOfSymbol_ReadAds].arrValue[uiLPWriteValueByArray_ReadAds] := CONCAT(stADSRead_ReadAds[udiActiveNumberOfSymbol_ReadAds].arrValue[uiLPWriteValueByArray_ReadAds],F_ToCHR(arrValueAfterRead_ReadAds[uiCounterArrayOfString_ReadAds]));
													IF arrValueAfterRead_ReadAds[uiCounterArrayOfString_ReadAds] = 0 AND stADSRead_ReadAds[udiActiveNumberOfSymbol_ReadAds].arrValue[uiLPWriteValueByArray_ReadAds] <> '' THEN	
														uiCounterArrayOfString_ReadAds := 31 * uiLPWriteValueByArray_ReadAds;	    
															EXIT; 
													ELSIF arrValueAfterRead_ReadAds[uiCounterArrayOfString_ReadAds] = 0 AND stADSRead_ReadAds[udiActiveNumberOfSymbol_ReadAds].arrValue[uiLPWriteValueByArray_ReadAds] = '' THEN 
														stADSRead_ReadAds[udiActiveNumberOfSymbol_ReadAds].arrValue[uiLPWriteValueByArray_ReadAds] := '#EMPTY#';
															uiCounterArrayOfString_ReadAds := 31 * uiLPWriteValueByArray_ReadAds;
																EXIT;	
													END_IF 
									END_FOR
								END_FOR 
				END_IF		END_IF
					//ARRAY OF TIME or ARRAY OF TIME OF DAY	
					IF FIND(Lynus_Standards.GVL_Communicator.arrInterfaceInfoAlVariables[byReadWriteArrayNumber,udiActiveNumberOfSymbol_ReadAds].sSymbolType,'OF TIME') <> 0 OR FIND(Lynus_Standards.GVL_Communicator.arrInterfaceInfoAlVariables[byReadWriteArrayNumber,udiActiveNumberOfSymbol_ReadAds].sSymbolType,'OF TIME_OF_DAY') <> 0 THEN
						stADSRead_ReadAds[udiActiveNumberOfSymbol_ReadAds].sFullSymbolName := Lynus_Standards.GVL_Communicator.arrInterfaceInfoAlVariables[byReadWriteArrayNumber,udiActiveNumberOfSymbol_ReadAds].sFullSymbolName;
							stADSRead_ReadAds[udiActiveNumberOfSymbol_ReadAds].arrValue := arrValueDefault_ReadAds;	
								IF Lynus_Standards.GVL_Communicator.arrInterfaceInfoAlVariables[byReadWriteArrayNumber,udiActiveNumberOfSymbol_ReadAds].uiSizeArray <= Lynus_Standards.Constants_Communicator.bySizeOfValueArray THEN  
									FOR uiLPWriteValueByArray_ReadAds := 1 TO Lynus_Standards.GVL_Communicator.arrInterfaceInfoAlVariables[byReadWriteArrayNumber,udiActiveNumberOfSymbol_ReadAds].uiSizeArray BY 1 DO
										arrCounterWriteValueInArray_ReadAds[1] := LIMIT(1,arrCounterWriteValueInArray_ReadAds[1],1600); arrCounterWriteValueInArray_ReadAds[2] := LIMIT(2,arrCounterWriteValueInArray_ReadAds[2],1600);
											arrCounterWriteValueInArray_ReadAds[3] := LIMIT(3,arrCounterWriteValueInArray_ReadAds[3],1600); arrCounterWriteValueInArray_ReadAds[4] := LIMIT(4,arrCounterWriteValueInArray_ReadAds[4],1600);
												stADSRead_ReadAds[udiActiveNumberOfSymbol_ReadAds].arrValue[uiLPWriteValueByArray_ReadAds] := UDINT_TO_STRING(SHL(BYTE_TO_UDINT(arrValueAfterRead_ReadAds[arrCounterWriteValueInArray_ReadAds[4]]),24) + SHL(BYTE_TO_UDINT(arrValueAfterRead_ReadAds[arrCounterWriteValueInArray_ReadAds[3]]),16) + SHL(BYTE_TO_UDINT(arrValueAfterRead_ReadAds[arrCounterWriteValueInArray_ReadAds[2]]),8) + BYTE_TO_UDINT(arrValueAfterRead_ReadAds[arrCounterWriteValueInArray_ReadAds[1]]));
										arrCounterWriteValueInArray_ReadAds[1] := arrCounterWriteValueInArray_ReadAds[1] + 4; arrCounterWriteValueInArray_ReadAds[2] := arrCounterWriteValueInArray_ReadAds[2] + 4;
											arrCounterWriteValueInArray_ReadAds[3] := arrCounterWriteValueInArray_ReadAds[3] + 4; arrCounterWriteValueInArray_ReadAds[4] := arrCounterWriteValueInArray_ReadAds[4] + 4;
									END_FOR 
								END_IF
					END_IF
				//ARRAY OF DATE or ARRAY OF DATE AND TIME
				IF FIND(Lynus_Standards.GVL_Communicator.arrInterfaceInfoAlVariables[byReadWriteArrayNumber,udiActiveNumberOfSymbol_ReadAds].sSymbolType,'OF DATE') <> 0 OR FIND(Lynus_Standards.GVL_Communicator.arrInterfaceInfoAlVariables[byReadWriteArrayNumber,udiActiveNumberOfSymbol_ReadAds].sSymbolType,'OF DATE_AND_TIME') <> 0 THEN
					stADSRead_ReadAds[udiActiveNumberOfSymbol_ReadAds].sFullSymbolName := Lynus_Standards.GVL_Communicator.arrInterfaceInfoAlVariables[byReadWriteArrayNumber,udiActiveNumberOfSymbol_ReadAds].sFullSymbolName;
						stADSRead_ReadAds[udiActiveNumberOfSymbol_ReadAds].arrValue := arrValueDefault_ReadAds;	
							IF Lynus_Standards.GVL_Communicator.arrInterfaceInfoAlVariables[byReadWriteArrayNumber,udiActiveNumberOfSymbol_ReadAds].uiSizeArray <= Lynus_Standards.Constants_Communicator.bySizeOfValueArray THEN  
								FOR uiLPWriteValueByArray_ReadAds := 1 TO Lynus_Standards.GVL_Communicator.arrInterfaceInfoAlVariables[byReadWriteArrayNumber,udiActiveNumberOfSymbol_ReadAds].uiSizeArray BY 1 DO
									arrCounterWriteValueInArray_ReadAds[1] := LIMIT(1,arrCounterWriteValueInArray_ReadAds[1],1600); arrCounterWriteValueInArray_ReadAds[2] := LIMIT(2,arrCounterWriteValueInArray_ReadAds[2],1600);
										arrCounterWriteValueInArray_ReadAds[3] := LIMIT(3,arrCounterWriteValueInArray_ReadAds[3],1600); arrCounterWriteValueInArray_ReadAds[4] := LIMIT(4,arrCounterWriteValueInArray_ReadAds[4],1600);
											uliValueDateTime_ReadAds := SHL(BYTE_TO_UDINT(arrValueAfterRead_ReadAds[arrCounterWriteValueInArray_ReadAds[4]]),24) + SHL(BYTE_TO_UDINT(arrValueAfterRead_ReadAds[arrCounterWriteValueInArray_ReadAds[3]]),16) + SHL(BYTE_TO_UDINT(arrValueAfterRead_ReadAds[arrCounterWriteValueInArray_ReadAds[2]]),8) + BYTE_TO_UDINT(arrValueAfterRead_ReadAds[arrCounterWriteValueInArray_ReadAds[1]]);
												uliValueDateTime_ReadAds := uliValueDateTime_ReadAds * 1000;	
													stADSRead_ReadAds[udiActiveNumberOfSymbol_ReadAds].arrValue[uiLPWriteValueByArray_ReadAds] := ULINT_TO_STRING(uliValueDateTime_ReadAds); 
									arrCounterWriteValueInArray_ReadAds[1] := arrCounterWriteValueInArray_ReadAds[1] + 4; arrCounterWriteValueInArray_ReadAds[2] := arrCounterWriteValueInArray_ReadAds[2] + 4;
										arrCounterWriteValueInArray_ReadAds[3] := arrCounterWriteValueInArray_ReadAds[3] + 4; arrCounterWriteValueInArray_ReadAds[4] := arrCounterWriteValueInArray_ReadAds[4] + 4;
								END_FOR 
							END_IF
				END_IF
					
			IF Lynus_Standards.GVL_Communicator.arrInterfaceInfoAlVariables[byReadWriteArrayNumber,udiActiveNumberOfSymbol_ReadAds].uiSizeArray <= Lynus_Standards.Constants_Communicator.bySizeOfValueArray AND iState_ReadAds = 5 THEN 
				arrCounterWriteValueInArray_ReadAds[1] := 0; arrCounterWriteValueInArray_ReadAds[2] := 0; arrCounterWriteValueInArray_ReadAds[3] := 0; 
					arrCounterWriteValueInArray_ReadAds[4] := 0; arrCounterWriteValueInArray_ReadAds[5] := 0; arrCounterWriteValueInArray_ReadAds[6] := 0; 
						arrCounterWriteValueInArray_ReadAds[7] := 0; arrCounterWriteValueInArray_ReadAds[8] := 0;
							uiCounterArrayOfString_ReadAds := 0;
								sStringFloat_ReadAds := ''; iFindPointFloat_ReadAds := 0; iPrecision_ReadAds := 0;
									iState_ReadAds := 6;
			 END_IF			
			
				IF timTimout_ReadAds.Q THEN iState_ReadAds := 200; END_IF
		
		ELSE
			IF udiActiveNumberOfSymbol_ReadAds < Lynus_Standards.GVL_Communicator.arrCounterVariableInArray[byReadWriteArrayNumber] AND udiNumberInProgress_ReadAds < udiNumberSizeValues_ReadAds THEN iState_ReadAds := -4; udiNumberInProgress_ReadAds := udiNumberInProgress_ReadAds + 1; END_IF
			IF (udiNumberInProgress_ReadAds >= udiNumberSizeValues_ReadAds AND iState_ReadAds = 5) THEN iState_ReadAds := -8; udiNumberInProgress_ReadAds := 0; END_IF
			IF udiActiveNumberOfSymbol_ReadAds >= Lynus_Standards.GVL_Communicator.arrCounterVariableInArray[byReadWriteArrayNumber] THEN iState_ReadAds := -8; udiActiveNumberOfSymbol_ReadAds := 0; udiNumberInProgress_ReadAds := 0; udiRestValueSymbolRead_ReadAds := 0; END_IF 
				//Timeout
				IF timTimout_ReadAds.Q THEN iState_ReadAds := 200; END_IF
		END_IF
	
	6://Check if the symbol exist
		byCounterWaitInStep_ReadAds := byCounterWaitInStep_ReadAds + 1;
			byCounterWaitInStep_ReadAds := LIMIT(1,byCounterWaitInStep_ReadAds,2);	
	
		IF byCounterWaitInStep_ReadAds = 1 THEN
			FOR udiLPCheckReadArrays_ReadAds := 1 TO udiNumberLoopHalf_ReadAds BY 1 DO
				IF stADSReadNew_ReadAds[udiLPCheckReadArrays_ReadAds].sFullSymbolName = Lynus_Standards.GVL_Communicator.arrInterfaceInfoAlVariables[byReadWriteArrayNumber,udiActiveNumberOfSymbol_ReadAds].sFullSymbolName THEN 
					iState_ReadAds := 7;																				//Symbol exist in the read array
				END_IF
			END_FOR
		END_IF
			IF byCounterWaitInStep_ReadAds = 2 AND udiNumberLoopFull_ReadAds <> udiNumberLoopHalf_ReadAds THEN
				FOR udiLPCheckReadArrays_ReadAds := (udiNumberLoopHalf_ReadAds + 1) TO udiNumberLoopFull_ReadAds BY 1 DO
					IF stADSReadNew_ReadAds[udiLPCheckReadArrays_ReadAds].sFullSymbolName = Lynus_Standards.GVL_Communicator.arrInterfaceInfoAlVariables[byReadWriteArrayNumber,udiActiveNumberOfSymbol_ReadAds].sFullSymbolName THEN 
						iState_ReadAds := 7;																			//Symbol exist in the read array
					END_IF
				END_FOR
			END_IF
		
				IF byCounterWaitInStep_ReadAds >= 2 AND iState_ReadAds = 6 THEN iState_ReadAds := 9; END_IF 			//Symbol not exist	
				
			//Timeout
			IF timTimout_ReadAds.Q THEN iState_ReadAds := 200; END_IF		
				
	7://Check if the value has changed
		byCounterWaitInStep_ReadAds := 0;
			bValueIsTheSame_ReadAds := FALSE;	
		
		FOR byLPCheckValueChange_ReadAds := 1 TO Lynus_Standards.Constants_Communicator.bySizeOfValueArray BY 1 DO
			IF stADSRead_ReadAds[udiActiveNumberOfSymbol_ReadAds].arrValue[byLPCheckValueChange_ReadAds] <> stADSReadNew_ReadAds[udiActiveNumberOfSymbol_ReadAds].arrValue[byLPCheckValueChange_ReadAds] THEN
				iState_ReadAds := 8;																																				//Value has changed
			ELSE		
				IF iState_ReadAds = 7 AND byLPCheckValueChange_ReadAds >= Lynus_Standards.Constants_Communicator.bySizeOfValueArray THEN iState_ReadAds := 10; bValueIsTheSame_ReadAds := TRUE; END_IF		//Value is the same
			END_IF 
		END_FOR	
		
			//Timeout
			IF timTimout_ReadAds.Q THEN iState_ReadAds := 200; END_IF	
		
	8://Symbol exist and Value has changed
		byCounterWaitInStep_ReadAds := byCounterWaitInStep_ReadAds + 1;
			byCounterWaitInStep_ReadAds := LIMIT(1,byCounterWaitInStep_ReadAds,2);
	
		IF byCounterWaitInStep_ReadAds = 1 THEN 
			FOR udiLPCheckReadArrays_ReadAds := 1 TO udiNumberLoopHalf_ReadAds BY 1 DO
				IF stADSRead_ReadAds[udiLPCheckReadArrays_ReadAds].sFullSymbolName = stADSReadNew_ReadAds[udiLPCheckReadArrays_ReadAds].sFullSymbolName THEN
					stADSReadNew_ReadAds[udiLPCheckReadArrays_ReadAds].arrValue := stADSRead_ReadAds[udiLPCheckReadArrays_ReadAds].arrValue;
				END_IF
			END_FOR
		END_IF	
			IF byCounterWaitInStep_ReadAds = 2 AND udiNumberLoopFull_ReadAds <> udiNumberLoopHalf_ReadAds THEN 
				FOR udiLPCheckReadArrays_ReadAds := (udiNumberLoopHalf_ReadAds + 1) TO udiNumberLoopFull_ReadAds BY 1 DO
					IF stADSRead_ReadAds[udiLPCheckReadArrays_ReadAds].sFullSymbolName = stADSReadNew_ReadAds[udiLPCheckReadArrays_ReadAds].sFullSymbolName THEN
						stADSReadNew_ReadAds[udiLPCheckReadArrays_ReadAds].arrValue := stADSRead_ReadAds[udiLPCheckReadArrays_ReadAds].arrValue;	
					END_IF
				END_FOR
			END_IF 
		
				IF byCounterWaitInStep_ReadAds >= 2 THEN iState_ReadAds := 10; END_IF			
		
			//Timeout
			IF timTimout_ReadAds.Q THEN iState_ReadAds := 200; END_IF
		
	9://Copy the new symbol in the array
		byCounterWaitInStep_ReadAds := 0;
			stADSReadNew_ReadAds := stADSRead_ReadAds;
				iState_ReadAds := 10;
			
	10://Write in Buffer if the send bus is busy or send a messege if the buffer is not empty
		byCounterWaitInStep_ReadAds := 0;
	
		IF NOT Lynus_Standards.GVL_Communicator.arrInterfaceInfoValueSendTo[byReadWriteArrayNumber].bBusy THEN	
			Lynus_Standards.GVL_Communicator.arrInterfaceInfoValueSendTo[byReadWriteArrayNumber].arrValue := arrValueDefault_ReadAds; 						//Clear send Interface if it is no message to send
				Lynus_Standards.GVL_Communicator.arrInterfaceInfoValueSendTo[byReadWriteArrayNumber].sSymbolUnit := ''; 
					Lynus_Standards.GVL_Communicator.arrInterfaceInfoValueSendTo[byReadWriteArrayNumber].sFullSymbolName := '';
						Lynus_Standards.GVL_Communicator.arrInterfaceInfoValueSendTo[byReadWriteArrayNumber].sSymbolType := '';
							IF fbBuffer_ReadAds.nCount > 0 THEN							
								iState_ReadAds := 11;														//Send a new messege from the buffer
							END_IF																			
		END_IF
			IF ((Lynus_Standards.GVL_Communicator.arrInterfaceInfoValueSendTo[byReadWriteArrayNumber].bBusy OR fbBuffer_ReadAds.nCount = 0) AND NOT bValueIsTheSame_ReadAds) THEN
				iState_ReadAds := 20;																		//Insert a new value in the buffer if the send bus is busy or no value is stored in the buffer
			ELSE
				IF iState_ReadAds = 10 THEN 																						
					iState_ReadAds := 100;																	//Value is the same
				END_IF																						
			END_IF
		
			//Timeout
			IF timTimout_ReadAds.Q THEN iState_ReadAds := 200; END_IF
	
	11://Read out a Value from the buffer for sending
		IF udiCounterReadBuffer_New_ReadAds <> fbBuffer_ReadAds.nCount AND fbBuffer_ReadAds.bOk THEN
			udiCounterReadBuffer_New_ReadAds := fbBuffer_ReadAds.nCount;
				IF fbBuffer_ReadAds.cbReturn <= 2000 THEN 
					FOR udiLPCheckReadBuffer_ReadAds := 1 TO fbBuffer_ReadAds.cbReturn BY 1 DO	
						IF byCounterValueReadOut_ReadAds = 0 AND arrBufferRead_ReadAds[udiLPCheckReadBuffer_ReadAds] <> 59 THEN sSymbolNameOutFromBuffer_ReadAds := CONCAT(sSymbolNameOutFromBuffer_ReadAds,F_ToCHR(arrBufferRead_ReadAds[udiLPCheckReadBuffer_ReadAds])); END_IF 
							IF arrBufferRead_ReadAds[udiLPCheckReadBuffer_ReadAds] = 59 THEN byCounterValueReadOut_ReadAds := byCounterValueReadOut_ReadAds + 1; END_IF
								byCounterValueReadOut_ReadAds := LIMIT(0,byCounterValueReadOut_ReadAds,Lynus_Standards.Constants_Communicator.bySizeOfValueArray);
									IF byCounterValueReadOut_ReadAds >= 1 AND arrBufferRead_ReadAds[udiLPCheckReadBuffer_ReadAds] <> 59 AND arrBufferRead_ReadAds[udiLPCheckReadBuffer_ReadAds] <> 0 THEN 
										arrValueOutFromBuffer_ReadAds[byCounterValueReadOut_ReadAds] := CONCAT(arrValueOutFromBuffer_ReadAds[byCounterValueReadOut_ReadAds],F_ToCHR(arrBufferRead_ReadAds[udiLPCheckReadBuffer_ReadAds])); 
									END_IF    	
					END_FOR				 
						IF arrBufferRead_ReadAds[udiLPCheckReadBuffer_ReadAds] = 0 THEN iState_ReadAds := 12; byCounterValueReadOut_ReadAds := 0; END_IF
				END_IF
		END_IF
		
			IF timTimout_ReadAds.Q THEN iState_ReadAds := 200; END_IF
	
	12://Write the Date on interface and start the sending
		byCounterWaitInStep_ReadAds := byCounterWaitInStep_ReadAds + 1;
			byCounterWaitInStep_ReadAds := LIMIT(1,byCounterWaitInStep_ReadAds,2);
	
		IF byCounterWaitInStep_ReadAds = 1 THEN 
			FOR udiLPCheckVarInfoBeforSending_ReadAds := 1 TO udiNumberLoopHalf_ReadAds BY 1 DO
				IF Lynus_Standards.GVL_Communicator.arrInterfaceInfoAlVariables[byReadWriteArrayNumber,udiLPCheckVarInfoBeforSending_ReadAds].sFullSymbolName = sSymbolNameOutFromBuffer_ReadAds THEN
					Lynus_Standards.GVL_Communicator.arrInterfaceInfoValueSendTo[byReadWriteArrayNumber].sFullSymbolName := sSymbolNameOutFromBuffer_ReadAds;
						Lynus_Standards.GVL_Communicator.arrInterfaceInfoValueSendTo[byReadWriteArrayNumber].sSymbolUnit := Lynus_Standards.GVL_Communicator.arrInterfaceInfoAlVariables[byReadWriteArrayNumber,udiLPCheckVarInfoBeforSending_ReadAds].sSymbolUnit;
							Lynus_Standards.GVL_Communicator.arrInterfaceInfoValueSendTo[byReadWriteArrayNumber].sSymbolType := Lynus_Standards.GVL_Communicator.arrInterfaceInfoAlVariables[byReadWriteArrayNumber,udiLPCheckVarInfoBeforSending_ReadAds].sSymbolType;
								Lynus_Standards.GVL_Communicator.arrInterfaceInfoValueSendTo[byReadWriteArrayNumber].arrValue := arrValueOutFromBuffer_ReadAds;
									Lynus_Standards.GVL_Communicator.arrInterfaceInfoValueSendTo[byReadWriteArrayNumber].bBusy := TRUE;
										iState_ReadAds := 13;
											EXIT;	
				END_IF 		 	   	
			END_FOR 	
		END_IF
			IF byCounterWaitInStep_ReadAds = 2 AND udiNumberLoopFull_ReadAds <> udiNumberLoopHalf_ReadAds THEN 
				FOR udiLPCheckVarInfoBeforSending_ReadAds := (udiNumberLoopHalf_ReadAds + 1) TO udiNumberLoopFull_ReadAds BY 1 DO
					IF Lynus_Standards.GVL_Communicator.arrInterfaceInfoAlVariables[byReadWriteArrayNumber,udiLPCheckVarInfoBeforSending_ReadAds].sFullSymbolName = sSymbolNameOutFromBuffer_ReadAds THEN
						Lynus_Standards.GVL_Communicator.arrInterfaceInfoValueSendTo[byReadWriteArrayNumber].sFullSymbolName := sSymbolNameOutFromBuffer_ReadAds;
							Lynus_Standards.GVL_Communicator.arrInterfaceInfoValueSendTo[byReadWriteArrayNumber].sSymbolUnit := Lynus_Standards.GVL_Communicator.arrInterfaceInfoAlVariables[byReadWriteArrayNumber,udiLPCheckVarInfoBeforSending_ReadAds].sSymbolUnit;
								Lynus_Standards.GVL_Communicator.arrInterfaceInfoValueSendTo[byReadWriteArrayNumber].sSymbolType := Lynus_Standards.GVL_Communicator.arrInterfaceInfoAlVariables[byReadWriteArrayNumber,udiLPCheckVarInfoBeforSending_ReadAds].sSymbolType;
									Lynus_Standards.GVL_Communicator.arrInterfaceInfoValueSendTo[byReadWriteArrayNumber].arrValue := arrValueOutFromBuffer_ReadAds;
										Lynus_Standards.GVL_Communicator.arrInterfaceInfoValueSendTo[byReadWriteArrayNumber].bBusy := TRUE;
											iState_ReadAds := 13;
												EXIT;	
					END_IF 		 	   	
				END_FOR 	
			END_IF
		
			IF timTimout_ReadAds.Q THEN iState_ReadAds := 200; END_IF
			
	13://Clear Read Buffer (conserve resources because the code must also work for small plc's)
		byCounterWaitInStep_ReadAds := 0;
			sSymbolNameOutFromBuffer_ReadAds := '';
				MEMCPY(ADR(arrBufferRead_ReadAds),ADR(arrBufferWriteReadDefault_ReadAds),SIZEOF(arrBufferRead_ReadAds));
					arrValueOutFromBuffer_ReadAds := arrValueDefault_ReadAds;
		
			iState_ReadAds := 10;
			
	20://Dim size from the values and symbol name befor can saving in buffer
		uiNumberValueSymbolSize_ReadAds := 0;
			byNumberOfValues_ReadAds_ReadAds := 0;
				byLenghSymbolName_ReadAds := 0;
		FOR byLPDimValueNumberASize_ReadAds := 1 TO Lynus_Standards.Constants_Communicator.bySizeOfValueArray BY 1 DO
			uiNumberValueSymbolSize_ReadAds := uiNumberValueSymbolSize_ReadAds + INT_TO_UINT(LEN(stADSReadNew_ReadAds[udiActiveNumberOfSymbol_ReadAds].arrValue[byLPDimValueNumberASize_ReadAds]));
				IF stADSReadNew_ReadAds[udiActiveNumberOfSymbol_ReadAds].arrValue[byLPDimValueNumberASize_ReadAds] <> '' THEN uiNumberValueSymbolSize_ReadAds := uiNumberValueSymbolSize_ReadAds + 1; END_IF 	
					IF stADSReadNew_ReadAds[udiActiveNumberOfSymbol_ReadAds].arrValue[byLPDimValueNumberASize_ReadAds] <> '' THEN byNumberOfValues_ReadAds_ReadAds := byNumberOfValues_ReadAds_ReadAds + 1; END_IF	
		END_FOR 	
			byLenghSymbolName_ReadAds := INT_TO_BYTE(LEN(stADSReadNew_ReadAds[udiActiveNumberOfSymbol_ReadAds].sFullSymbolName));
				uiNumberValueSymbolSize_ReadAds := uiNumberValueSymbolSize_ReadAds + byLenghSymbolName_ReadAds + 1;
		
			IF byNumberOfValues_ReadAds_ReadAds <= Lynus_Standards.Constants_Communicator.bySizeOfValueArray THEN
				FOR byLPDimLenghValues_ReadAds := 1 TO byNumberOfValues_ReadAds_ReadAds BY 1 DO
					arrLenghEachValue_ReadAds[byLPDimLenghValues_ReadAds] := INT_TO_BYTE(LEN(stADSReadNew_ReadAds[udiActiveNumberOfSymbol_ReadAds].arrValue[byLPDimLenghValues_ReadAds]));	
				END_FOR 
			END_IF
	
		IF byNumberOfValues_ReadAds_ReadAds <= Lynus_Standards.Constants_Communicator.bySizeOfValueArray AND byNumberOfValues_ReadAds_ReadAds >= 1 AND uiNumberValueSymbolSize_ReadAds <> 0 THEN iState_ReadAds := 21; END_IF
		
			IF timTimout_ReadAds.Q THEN iState_ReadAds := 200; END_IF
			
	21://String to Ascii Symbol Name and values
		IF byLenghSymbolName_ReadAds <= 49 THEN
			FOR byLPSymbolNameToAscii_ReadAds := 1 TO byLenghSymbolName_ReadAds BY 1 DO
				arrSymbolName_ReadAds[byLPSymbolNameToAscii_ReadAds] := F_ToASC(MID(stADSReadNew_ReadAds[udiActiveNumberOfSymbol_ReadAds].sFullSymbolName,1,byLPSymbolNameToAscii_ReadAds));
			END_FOR 
		END_IF
			IF byLenghSymbolName_ReadAds < 49 THEN arrSymbolName_ReadAds[byLenghSymbolName_ReadAds + 1] := F_ToASC(';'); END_IF  	
		
		IF byNumberOfValues_ReadAds_ReadAds <= Lynus_Standards.Constants_Communicator.bySizeOfValueArray THEN 
			FOR byLPValueNameToAscii_1_ReadAds := 1 TO byNumberOfValues_ReadAds_ReadAds BY 1 DO
				IF arrLenghEachValue_ReadAds[byLPValueNameToAscii_1_ReadAds] <= 31 THEN 
					FOR byLPValueNameToAscii_2_ReadAds := 1 TO arrLenghEachValue_ReadAds[byLPValueNameToAscii_1_ReadAds] BY 1 DO
						arrValueName_ReadAds[byLPValueNameToAscii_1_ReadAds,byLPValueNameToAscii_2_ReadAds] := F_ToASC(MID(stADSReadNew_ReadAds[udiActiveNumberOfSymbol_ReadAds].arrValue[byLPValueNameToAscii_1_ReadAds],1,byLPValueNameToAscii_2_ReadAds));
					END_FOR
				END_IF
					arrValueName_ReadAds[byLPValueNameToAscii_1_ReadAds,byLPValueNameToAscii_2_ReadAds] := F_ToASC(';'); 			
			END_FOR 
		END_IF 
		
		IF byLenghSymbolName_ReadAds <= 49 AND byNumberOfValues_ReadAds_ReadAds <= Lynus_Standards.Constants_Communicator.bySizeOfValueArray AND arrLenghEachValue_ReadAds[byNumberOfValues_ReadAds_ReadAds] <= 31 THEN iState_ReadAds := 22; END_IF
		
			IF timTimout_ReadAds.Q THEN iState_ReadAds := 200; END_IF	
			
	22://Prepare Write array for Buffer
		IF byLenghSymbolName_ReadAds <= 48 THEN
			FOR uiLPWriteByteValueInArray_ReadAds := 1 TO (byLenghSymbolName_ReadAds + 1) BY 1 DO
				arrBufferWrite_ReadAds[uiLPWriteByteValueInArray_ReadAds] := arrSymbolName_ReadAds[uiLPWriteByteValueInArray_ReadAds];
			END_FOR 
		END_IF
		
		IF byLenghSymbolName_ReadAds <= 48 THEN	iState_ReadAds := 23; END_IF
			
			IF timTimout_ReadAds.Q THEN iState_ReadAds := 200; END_IF
	
	23://Prepare Write array for Buffer
		uiValueForLoopStart_ReadAds := uiLPWriteByteValueInArray_ReadAds;
			byValueInTurn_ReadAds := byValueInTurn_ReadAds + 1;
				byValueInTurn_ReadAds := LIMIT(1,byValueInTurn_ReadAds,Lynus_Standards.Constants_Communicator.bySizeOfValueArray);
					uiValueForLoopStop_ReadAds := arrLenghEachValue_ReadAds[byValueInTurn_ReadAds] + uiValueForLoopStart_ReadAds;
						byCounterValue_ReadAds := 0;
							
							IF uiValueForLoopStart_ReadAds >= 1 AND uiValueForLoopStart_ReadAds <= 2000 AND uiValueForLoopStop_ReadAds >= 1 AND uiValueForLoopStop_ReadAds <= 2000 THEN 
								FOR uiLPWriteByteValueInArray_ReadAds := uiValueForLoopStart_ReadAds TO uiValueForLoopStop_ReadAds BY 1 DO
									byCounterValue_ReadAds :=  byCounterValue_ReadAds + 1;
										byCounterValue_ReadAds := LIMIT(1,byCounterValue_ReadAds,31);	
											arrBufferWrite_ReadAds[uiLPWriteByteValueInArray_ReadAds] := arrValueName_ReadAds[byValueInTurn_ReadAds,byCounterValue_ReadAds];
								END_FOR 
							END_IF
		
		IF byValueInTurn_ReadAds >= byNumberOfValues_ReadAds_ReadAds AND uiValueForLoopStart_ReadAds >= 1 AND uiValueForLoopStart_ReadAds <= 2000 AND uiValueForLoopStop_ReadAds >= 1 AND uiValueForLoopStop_ReadAds <= 2000 THEN 
			iState_ReadAds := 24; 
				uiValueForLoopStart_ReadAds := 0;
					byValueInTurn_ReadAds := 0;
						uiValueForLoopStop_ReadAds := 0;
							byCounterValue_ReadAds := 0;			
		END_IF
			
			IF timTimout_ReadAds.Q THEN iState_ReadAds := 200; END_IF

	24://Write Value in Buffer
		iState_ReadAds := 25; 
				
	25://Check if the new value is stored in the buffer
		IF fbBuffer_ReadAds.bOk AND fbBuffer_ReadAds.nCount <> udiCounterReadBuffer_New_ReadAds THEN udiCounterReadBuffer_New_ReadAds := fbBuffer_ReadAds.nCount; iState_ReadAds := 26; END_IF  	
			
			IF timTimout_ReadAds.Q THEN iState_ReadAds := 200; END_IF
		
	26://Clear the Write Buffer (conserve resources because the code must also work for small plc's)
		MEMCPY(ADR(arrBufferWrite_ReadAds),ADR(arrBufferWriteReadDefault_ReadAds),SIZEOF(arrBufferWrite_ReadAds));
		
			iState_ReadAds := 100;

	100://Check for other variable
		//Next symbol
		IF udiActiveNumberOfSymbol_ReadAds < Lynus_Standards.GVL_Communicator.arrCounterVariableInArray[byReadWriteArrayNumber] AND udiNumberInProgress_ReadAds < udiNumberSizeValues_ReadAds THEN iState_ReadAds := -4; udiNumberInProgress_ReadAds := udiNumberInProgress_ReadAds + 1; END_IF
			//Start with the next 10 Variables
			IF (udiNumberInProgress_ReadAds >= udiNumberSizeValues_ReadAds AND iState_ReadAds = 100) THEN 
				iState_ReadAds := -8; 
					udiNumberInProgress_ReadAds := 0;
			END_IF	
				//Start from New with the first 10 Variables 	
				IF udiActiveNumberOfSymbol_ReadAds >= Lynus_Standards.GVL_Communicator.arrCounterVariableInArray[byReadWriteArrayNumber] THEN
					iState_ReadAds := -8; 
						udiActiveNumberOfSymbol_ReadAds := 0;
							udiNumberInProgress_ReadAds := 0;
								udiRestValueSymbolRead_ReadAds := 0;
						 			bFirstReadCycleDone_ReadAds := TRUE; 
				END_IF			
			
			bError_ReadAds := FALSE;
				uiInternError_ReadAds := 0;
			
			IF timTimout_ReadAds.Q THEN iState_ReadAds := 200; END_IF
				
	200://Error
		bError_ReadAds := TRUE; fbADSREADWRITE_ReadAds.WRTRD := FALSE; bValueIsTheSame_ReadAds := FALSE; 
			udiActiveNumberOfSymbol_ReadAds := 0; byCounterWaitInStep_ReadAds := 0; udiNumberInProgress_ReadAds := 0; udiRestValueSymbolRead_ReadAds := 0;
		
		//Clear the write Buffer befor go to step 0 (conserve resources because the code must also work for small plc's)
		MEMCPY(ADR(arrBufferWrite_ReadAds),ADR(arrBufferWriteReadDefault_ReadAds),SIZEOF(arrBufferWrite_ReadAds));
		
		//Clear the read Buffer befor go to step 0 (conserve resources because the code must also work for small plc's)
		sSymbolNameOutFromBuffer_ReadAds := '';
			MEMCPY(ADR(arrBufferRead_ReadAds),ADR(arrBufferWriteReadDefault_ReadAds),SIZEOF(arrBufferRead_ReadAds));
				arrValueOutFromBuffer_ReadAds := arrValueDefault_ReadAds;
			
		//Count up when an error has occurred
		byErrorCounter_ReadAds := byErrorCounter_ReadAds + 1;		
				
			iState_ReadAds := 300;
	
	300://Wait in Error and clear the rest from the read and write buffer (conserve resources because the code must also work for small plc's)
		byCounterWaitInStep_ReadAds := byCounterWaitInStep_ReadAds + 1;
	
			//Restart new from in Step -8. No Reset from the complete System
			IF byCounterWaitInStep_ReadAds > 10 AND byErrorCounter_ReadAds <= 10 THEN byCounterWaitInStep_ReadAds := 0; iState_ReadAds := -8; END_IF
				//Restart new from in Step -10. Reset from the complete System after to much Errors
				IF byCounterWaitInStep_ReadAds > 10 AND byErrorCounter_ReadAds > 10 THEN 
						byCounterWaitInStep_ReadAds := 0; 
							//Reset Read Steps and start from new
							iState_ReadAds := -10;
								//Reset Write Steps and start from new
								iState_WriteAds := -2;
									byErrorCounter_ReadAds := 0; 
				END_IF
	
END_CASE	

//Resetting the error counter after not being in the error step for 30 min
timResetErrorCounter_ReadAds(IN:= byErrorCounter_ReadAds <> 0, PT:= T#30M, Q=> , ET=> );
	IF timResetErrorCounter_ReadAds.Q THEN byErrorCounter_ReadAds := 0; END_IF 

//Read Out Variable by ADS
fbADSREADWRITE_ReadAds(
	NETID:= fbNedID.AddrString, 
	PORT:= uiPort, 
	IDXGRP:= 16#F080, 
	IDXOFFS:= udiNumberSizeValues_ReadAds, 
	WRITELEN:= , 
	READLEN:= udiSizeReq_ReadAds, 
	SRCADDR:= , 
	DESTADDR:= ADR(arrValueRead_ReadAds), 
	WRTRD:= , 
	TMOUT:= T#5S, 
	BUSY=> , 
	ERR=> , 
	ERRID=> );

FPErrorReadWrite_ReadAds(CLK:= fbADSREADWRITE_ReadAds.ERR, Q=> );	
	
//Buffer Read Value from ADS
FPWriteValueToBufferStep25_ReadAds(CLK:= iState_ReadAds = 24, Q=> );
FPReadValueToBufferStep11_ReadAds(CLK:= iState_ReadAds = 11, Q=> );

IF FPReadValueToBufferStep11_ReadAds.Q THEN fbBuffer_ReadAds.A_RemoveHead(); END_IF
IF FPWriteValueToBufferStep25_ReadAds.Q THEN fbBuffer_ReadAds.A_AddTail(); END_IF

//Reset the Buffer after a Buffer Overflow
IF fbBuffer_ReadAds.nCount <> 0 AND NOT fbBuffer_ReadAds.bOk THEN timResetBuffer_ReadAds.IN := TRUE; ELSE timResetBuffer_ReadAds.IN := FALSE; END_IF
	timResetBuffer_ReadAds(IN:= , PT:= T#40S, Q=> , ET=> );
		IF timResetBuffer_ReadAds.Q THEN fbBuffer_ReadAds.A_Reset(); END_IF

fbBuffer_ReadAds(
	pWrite:= ADR(arrBufferWrite_ReadAds), 
	cbWrite:= uiNumberValueSymbolSize_ReadAds, 
	pRead:= ADR(arrBufferRead_ReadAds), 
	cbRead:= SIZEOF(arrBufferRead_ReadAds), 
	pBuffer:= ADR(arrBufferADSRead_ReadAds), 
	cbBuffer:= SIZEOF(arrBufferADSRead_ReadAds), 
	bOk=> Lynus_Standards.GVL_Communicator.arrInterfaceInfoValueSendTo[byReadWriteArrayNumber].bBufferOK, 
	nCount=> Lynus_Standards.GVL_Communicator.arrInterfaceInfoValueSendTo[byReadWriteArrayNumber].udiCountBuffer, 
	cbSize=> , 
	cbReturn=> );

END_IF
	
//Busy
IF iState_ReadAds >= -8 OR iState_WriteAds >= 0 THEN bBusy := TRUE; ELSE bBusy := FALSE; END_IF
	
//Error
IF (bError_ReadAds AND iState_ReadAds <> - 10 AND iState_ReadAds <> - 9) OR (bError_WriteAds AND iState_WriteAds <> - 1 AND iState_WriteAds <> - 2) THEN fbErrorCodes.bErrorIntern := TRUE; ELSE fbErrorCodes.bErrorIntern := FALSE; END_IF

IF fbADSREADWRITE_ReadAds.ERR OR fbADSREADWRITE_WriteAds.ERR OR fbADSWrite_WriteAds.ERR THEN fbErrorCodes.bErrorADS := TRUE; END_IF

IF fbADSREADWRITE_ReadAds.ERR THEN fbErrorCodes.udiErrorCodeADS := fbADSREADWRITE_ReadAds.ERRID; END_IF
IF fbADSREADWRITE_WriteAds.ERR THEN fbErrorCodes.udiErrorCodeADS := fbADSREADWRITE_WriteAds.ERRID; END_IF
IF fbADSWrite_WriteAds.ERR THEN fbErrorCodes.udiErrorCodeADS := fbADSWrite_WriteAds.ERRID; END_IF

IF NOT fbADSREADWRITE_ReadAds.ERR AND NOT fbADSREADWRITE_ReadAds.BUSY AND NOT
	fbADSREADWRITE_WriteAds.ERR AND NOT fbADSREADWRITE_WriteAds.BUSY AND NOT fbADSWrite_WriteAds.ERR AND NOT fbADSWrite_WriteAds.BUSY THEN 
		fbErrorCodes.bErrorADS := FALSE;
			fbErrorCodes.udiErrorCodeADS := 0; 
END_IF 	     
	
fbErrorCodes(
	bErrorADS:= , 
	bErrorIntern:= , 
	udiErrorCodeADS:= , 
	udiErrorCodesInternRead:= uiInternError_ReadAds, 
	udiErrorCodesInternWrite:= uiInternError_WriteAds, 
	udiErrorCodeADS_Out=> udiErrorCodeOut, 
	bError=> bError, 
	eErrorReadWrite_Out=> eErrorReadWrite_Out);

END_FUNCTION_BLOCK

// ---- FB/FB_VarInfo.TcPOU
{attribute 'hide_all_locals'}
FUNCTION_BLOCK FB_VarInfo
VAR_INPUT
	bReadInfo						: BOOL;																									//Manually start to read the information of plc variables with a rising edge
	eTMCFile						: eSelectTMCFile;																						//Option to select the TMC file if Structs, Functionblocks or Enums are in using in the plc Code to push in the Cloud
	eSavePositionTMCFile			: eSavePositionOnPLC;																					//Choose the Saveposition from the TMC File
END_VAR
VAR_OUTPUT
	udiCounterFoundVariables		: UDINT;																								//Counter of found variables on the plc with the comment for cloud service
	bError							: BOOL;																									//Error flag
	bBusy							: BOOL;																									//Busy flag
	byProgress						: BYTE;																									//Progress from the function in 0-100%
	udiErrorCodeOut					: UDINT;																								//Error ID, it is a internal Beckhoff Error		
	eErrorVarInfo_Out				: eErrorVarInfo;																						//Enum with Error from the Var Info function	
	sVarWithError					: STRING(255);																							//Variable with Error												
END_VAR
VAR
	fbNedID							: FB_GetLocalAmsNetId := (bExecute := TRUE);															//Functionblock to detect the AMSNetId form the local plc
	fbADSRead						: ADSREAD;																								//Functionblock AMSREAD
	fbADSInfoSubItem				: ADSRDWRT;																								//Function to read the Infos from the SubItems
	fbTaskIndex						: GETCURTASKINDEX;																						//Task Index
	fbADSErrorCodes					: FB_VarInfo_ErrorCodes;																				//Function Block for ADS Error Codes
	fbParseDocument					: FB_ParsDocument;																						//Function to parse the TMC File from Information
	stSymbolUploadInfo				: ST_Symbol_Upload_Info;																				//Infos about the numbers and size of the variables
	stADSSymbolUpload				: ST_Symbol_Upload_Raw; 																				//Infos from the plc variable
	stADSVarInfo					: ST_Var_Info;																							//Var info
	stDataSubItems					: ST_Symbol_Info_SubItem;																				//Data with Infos from the SubItems
	FPError							: R_TRIG;																								//Internal rising edge 
	FPErrorADSInfoSubItem			: R_TRIG;																								//Internal rising edge 
	FPErrorParse					: R_TRIG;																								//Internal rising edge
	FPRead							: R_TRIG;																								//Internal rising edge 
	FPBusy							: R_TRIG;																								//Internal rising edge 
	FPTimoutTime					: R_TRIG;																								//Internal rising edge
	FNBusy							: F_TRIG;																								//Internal falling edge 
	timTimout						: TON;																									//Timer for Timeout
	eTMCFile_Int					: eSelectTMCFile;																						//Internal Enum to compare with the Input Enum to detected a change of the value 
	eSavePositionTMCFile_Int		: eSavePositionOnPLC;																					//Internal Enum to compare with the Input Enum to detected a change of the value
	bBusyInt						: BOOL;																									//Internal Busy flag
	bErrorIntern					: BOOL;																									//Intern error flag
	bNoStandardDatatypeDetected		: BOOL;																									//True if it is not a standart datatype
	bFirstCykle						: BOOL;																									//True if plc cycle begin
	bStringDetected					: BOOL;																									//True if the symbol is a string
	bSymbolInTMCFileFound			: BOOL;																									//Is true if in TMC File Symbols are found
	bNewStart						: BOOL;																									//Start new Scanning Session
	bDataTypeIsStandart				: BOOL;																									//True if the Symbol is a Standart Type
	bLastCycle						: BOOL;																									//True when the function check the last symbol in Subitems
	byLPClearArraySubItemInfo		: BYTE;																									//Loop tp clear the Info from the Subitems
	byCounterWaitInStep				: BYTE;																									//Counter to wait in each step of statemaschine
	byCounterNumberFuctionInfo		: BYTE;																									//Counter with fuction Info
	byCounterNumberFuctionReadWrite	: BYTE;																									//Counter with fuction read write
	byCounterSendReceiveFunction	: BYTE;																									//Counter with fuction send/receive
	byCounterWriteDataToGV			: BYTE;																									//Counter to Write Global Data
	byArrayInProgress				: BYTE;																									//Array in progress where the values are written in 
	byProgressClearVarInterface		: BYTE;																									//Progress to clear Var Interface
	byProgressParseDocument			: BYTE;																									//Progress Parse TMC File
	byProgressSubItems				: BYTE;																									//Progress SubItems
	byProgressCopyArray				: BYTE;																									//Progress Copy Array
	byLPFindPoints					: BYTE;																									//Loop to find points in Symbol Name (Step 23)
	byPointsFound					: BYTE;																									//Points found in the Full Symbol name to ckeck big datatypes (Step 23)
	uiSizeArray						: UINT;																									//Array Size 
	uiValueLower					: UINT;																									//Lower value from array size
	uiValueHigher					: UINT;																									//Higher value from array size
	uiPort							: UINT;																									//Port from TC3
	uiStateRead						: UINT;																									//Variable from the statemschine
	uiStateRead_CP					: UINT;																									//Comparison variable
	uiStateCheckComment				: UINT;																									//Variable from statemaschine to check comment
	uiStateCheckEnum				: UINT;																									//State maschine to check if the symbol is a enum
	uiStateVarToGVInterface			: UINT;																									//State maschine to write var on globale interface 
	uiCounterCheckSymbolsTMCFile	: UINT;																									//Counter for checked Symbols in TMC File
	uiLPClearOutputArray			: UINT;																									//Loop to clear the Output Array
	udiLengthTo_0					: UDINT;																								//Variable that includes the index from start to the next 0 in the array of the variable infos
	udiFactortLP					: UDINT;																								//Factor that was detected for next atart of information in the array of the variable infos
	udiLPSearch_0					: UDINT;																								//Loop for search next 0 in the array of the variable infos
	udiCounterClearOutputArray		: UDINT;																								//Counter for clear Output Array befor new read session
	udiCounterWriteDataToGV			: UDINT;																								//Counter to Write default in Global Data
	udiErrorIntern					: UDINT;																								//Intern error Code
	udiCounterOnlineChange			: UDINT;																								//Counter Online Change
	udiCycleTime					: UDINT;																								//Cycle Time
	udiCounterSymbol				: UDINT;																								//Counter from 0 to max symbols on plc
	udiCounterRestSymbol			: UDINT;																								//Rest of not used symbols for next position in array
	udiNumbersForArray				: UDINT;																								//Number of Symbols per array
	udiCounterFillSymbolArray		: UDINT;																								//Counter to fill the values in the right position in array
	udiLPFillSymbolsInArray			: UDINT;																								//Loop to fill the values in array
	udiCounterCheckNoStandartType	: UDINT;																								//Counter to check in the inforamtion for no standart data types
	udiNumberOfNoStandartDataType	: UDINT;																								//Numbers from no standart data types in the informations
	udiCounterCopyArrayToFinalArray	: UDINT;																								//Counter to Copy the Arrays
	udiCounterFoundVariablesInt		: UDINT;																								//Internal Counter of found variables on the plc with the comment for cloud service
	rWaitInStep						: REAL;																									//Wait Value, to wait in one step about the state maschine
	uliSizeOfString					: ULINT;																								//Size of the String
	sFullSymbolNameToCkeck			: STRING(48);																							//Full Symbol name to check points for big data type (Step 23)
	sCommentInfos					: STRING(255);																							//Comment Infos
	arrADSInfoSubItem				: ARRAY[1..12] OF BYTE;																					//Array wit Infos from the SubItems
	arrFirstCounterToCheckSubItems	: ARRAY[1..4] OF UDINT;																					//Counter to copy Content from Array to a other Array
	arrSecondCounterToCheckSubItems	: ARRAY[1..2] OF UDINT;																					//Counter to copy Content from Array to a other Array
	arrSymbols						: ARRAY[0..Lynus_Standards.Constants_Communicator.udiArraySizeSymbols] OF BYTE;							//Raw information from plc variable
	arrFind							: ARRAY[1..4] OF INT;																					//Array for find symbols
	arrVarInfos						: ARRAY[1..Lynus_Standards.Constants_Communicator.udiArraySizeMarkedSymobls] OF ST_Var_Info_EX;			//Infos from each plc variable
	arrAllVarInfosForGV				: ARRAY[1..Lynus_Standards.Constants_Communicator.udiArraySizeMarkedSymobls] OF ST_Var_Info_EX_All;		//Infos from each plc variable after adding all the Subitems 
END_VAR

//Creator : Kai Ebensperger
//Company : Lynus AG
//Updated : M.Schwarzmann, EfficientIO
//Date : 08.06.2022
//Version : 2.0.0.1

//Function how can read the infos of all standart plc variables and arrays in the local plc
//Al standart variables they are signed by //{#lynus.ag#()} are stored for read and write
//Strings are limited at 30 characters
//Arrays are limited at a size of 1, because belonging in the cloud is difficult
//2-3 dimensional array at this version not working
//If its a ADS Error or a internal Error the fuction produce an error
//If you want to work with Structs, Enums or FB the TMC File fromt the plc project is needed. 
//Use this Path for the TMC File = C:\TwinCAT\3.1\Config\TMC\ for Win7 or higher or Hard Disk\TwinCAT\3.1\Config\TMC\ for Win CE
//Every Struct or FB can have a other 1 Subitem. More is not allowed. 
//With structures, however, it depends on whether they are called in an FB or directly in the program.
//FB calls in Structs is not allowed.
//Arrays from FB's, Structs or Enums are not allowed.
//Every Symbol in a Big Data Type (FB or Struct) is 1 Symbol in the Array List for the GVL.
//Every Big Data Symbol can have max 50 Subitems
//At the last every Big Data Symbol can have max 50 Subitems with all Subitems that are included

//Read TC3 Port
uiPort := TwinCAT_SystemInfoVarList._AppInfo.AdsPort;

//Read AMS Net ID from the local plc
fbNedID();
	IF (NOT fbNedID.bBusy) AND NOT fbNedID.bError THEN fbNedID.bExecute := FALSE; END_IF

//TaskIndex
fbTaskIndex(index=> );
	udiCycleTime := TwinCAT_SystemInfoVarList._TaskInfo[fbTaskIndex.index].CycleTime / 10000;
	
//Wait in Step min 2 x Cycle Time for ADS Response
rWaitInStep := STRING_TO_REAL(LREAL_TO_FMTSTR((UDINT_TO_LREAL(udiCycleTime) / 10) * 2,0,FALSE)); 
	rWaitInStep := LIMIT(2,rWaitInStep,20);

//Timer for timeout
FPTimoutTime(CLK:= uiStateRead = 1, Q=> );
	IF FPTimoutTime.Q THEN timTimout.PT := (T#25S * (udiCycleTime + (Lynus_Standards.Constants_Communicator.udiArraySizeMarkedSymobls / 100))) / 4; END_IF
		timTimout(IN:= uiStateRead <> uiStateRead_CP AND TwinCAT_SystemInfoVarList._AppInfo.OnlineChangeCnt = udiCounterOnlineChange, PT:= , Q=> , ET=> );
			IF uiStateRead = 100 OR uiStateRead = 0 THEN timTimout.PT := T#5S; END_IF
				IF uiStateRead > 100 THEN timTimout.PT := T#30S; END_IF 

//Dont change the Enums if the Function is running
IF uiStateRead = 0 THEN eTMCFile_Int := eTMCFile; eSavePositionTMCFile_Int := eSavePositionTMCFile; END_IF			
			
//Start State Maschine
FPRead(CLK:= bReadInfo, Q=> );
	IF TwinCAT_SystemInfoVarList._TaskInfo[fbTaskIndex.index].FirstCycle THEN bFirstCykle := TRUE; END_IF
	
IF (NOT fbNedID.bExecute AND uiStateRead = 0 AND NOT fbADSRead.BUSY AND FPRead.Q) OR
	(NOT fbNedID.bExecute AND udiCounterOnlineChange <> TwinCAT_SystemInfoVarList._AppInfo.OnlineChangeCnt AND uiStateRead = 2 AND NOT fbADSRead.BUSY) OR 
		(NOT fbNedID.bExecute AND udiCounterOnlineChange <> TwinCAT_SystemInfoVarList._AppInfo.OnlineChangeCnt AND uiStateRead = 0 AND NOT fbADSRead.BUSY) OR 
			(NOT fbNedID.bExecute AND udiCounterOnlineChange <> TwinCAT_SystemInfoVarList._AppInfo.OnlineChangeCnt AND uiStateRead = 110 AND NOT fbADSRead.BUSY) OR 
				(NOT fbNedID.bExecute AND udiCounterOnlineChange <> TwinCAT_SystemInfoVarList._AppInfo.OnlineChangeCnt AND uiStateRead = 111 AND NOT fbADSRead.BUSY) OR 
					(NOT fbNedID.bExecute AND udiCounterOnlineChange <> TwinCAT_SystemInfoVarList._AppInfo.OnlineChangeCnt AND uiStateRead = 112 AND NOT fbADSRead.BUSY) OR 
						(NOT fbNedID.bExecute AND bFirstCykle) THEN 
							uiStateRead := 0;
								bNewStart := TRUE;
END_IF
	
IF uiStateRead = 0 AND bNewStart THEN udiCounterOnlineChange := TwinCAT_SystemInfoVarList._AppInfo.OnlineChangeCnt; bFirstCykle := FALSE; END_IF	

//State Maschine 

CASE uiStateRead OF
	
	0: //Init and set default Values
		bBusy := FALSE;
			bBusyInt := FALSE;
		
		fbADSRead.READ := FALSE; byCounterWaitInStep := 0; udiLengthTo_0 := 0; udiFactortLP := 0; fbADSInfoSubItem.WRTRD := FALSE;					
			arrFind[1] := 0; arrFind[2] := 0; arrFind[3] := 0; arrFind[4] := 0; uiStateCheckComment := 0; udiCounterSymbol := 0; byProgressClearVarInterface := 0; byProgressCopyArray := 0; udiCounterCopyArrayToFinalArray := 0; 
				sCommentInfos := '';
					uiSizeArray := 0; uiValueHigher := 0; uiValueLower := 0; uliSizeOfString := 0; udiCounterCheckNoStandartType := 0; bNoStandardDatatypeDetected := FALSE; bStringDetected := FALSE;
						fbParseDocument.bRead := FALSE; bSymbolInTMCFileFound := FALSE; bDataTypeIsStandart := FALSE; bLastCycle := FALSE; uiCounterCheckSymbolsTMCFile := 0; udiCounterClearOutputArray := 0; uiStateCheckEnum := 0;
							byProgressSubItems := 0; byProgressParseDocument := 0; uiStateRead_CP := 0; arrFirstCounterToCheckSubItems[1] := 0; arrFirstCounterToCheckSubItems[2] := 0; arrFirstCounterToCheckSubItems[3] := 0;
								arrFirstCounterToCheckSubItems[4] := 0; arrSecondCounterToCheckSubItems[1] := 0; arrSecondCounterToCheckSubItems[2] := 0; stDataSubItems.udiSubItemGroup := 0; stDataSubItems.udiSubItemOffset := 0; stDataSubItems.udiSubItemSize := 0;
									sFullSymbolNameToCkeck := ''; byPointsFound := 0;								
																							
		IF fbParseDocument.bBusy THEN fbParseDocument.bStop := TRUE; END_IF
																						
		IF bNewStart THEN
			byCounterNumberFuctionInfo := 0;
				byCounterNumberFuctionReadWrite := 0; 
					byCounterSendReceiveFunction := 0;
						byProgress := 0;	
							uiStateRead := 1000;
								bNewStart := FALSE;	
		END_IF
	
	1: //Read the length of the Variable declaration and set Default und Arrays
		bBusy := TRUE;
			bBusyInt := TRUE;
				Lynus_Standards.GVL_Communicator.bInfoAlVariablesOK := FALSE;
					byCounterNumberFuctionInfo := 0;
						byCounterNumberFuctionReadWrite := 0;
							byCounterSendReceiveFunction := 0;
								udiNumberOfNoStandartDataType := 0;
	
		//Clear Arrays
		IF udiCounterClearOutputArray < udiCounterFoundVariablesInt THEN udiCounterClearOutputArray := udiCounterClearOutputArray + 1; END_IF
			udiCounterClearOutputArray := LIMIT(1,udiCounterClearOutputArray,Lynus_Standards.Constants_Communicator.udiArraySizeMarkedSymobls);					
							
		IF udiCounterClearOutputArray <= udiCounterFoundVariablesInt THEN  
			arrVarInfos[udiCounterClearOutputArray].sSymbolName := '';
				arrVarInfos[udiCounterClearOutputArray].sSymbolType := '';
					arrVarInfos[udiCounterClearOutputArray].udiGroup := 0;
						arrVarInfos[udiCounterClearOutputArray].udiOffset := 0;
							arrVarInfos[udiCounterClearOutputArray].udiFlags := 0;
								arrVarInfos[udiCounterClearOutputArray].udiSize := 0;
									arrVarInfos[udiCounterClearOutputArray].uiSizeArray := 0;
										arrVarInfos[udiCounterClearOutputArray].uiTypeLength := 0;	
											arrVarInfos[udiCounterClearOutputArray].sFullSymbolName := '';
												arrVarInfos[udiCounterClearOutputArray].sProjectName := '';
													arrVarInfos[udiCounterClearOutputArray].sSymbolUnit := '';
														arrVarInfos[udiCounterClearOutputArray].sAdsDataType := '';
															arrVarInfos[udiCounterClearOutputArray].bNoStandardDatatypeDetected := FALSE;	
																FOR uiLPClearOutputArray := 1 TO Lynus_Standards.Constants_Communicator.uiArraySizeOfMarkedSubItems BY 1 DO
																	arrVarInfos[udiCounterClearOutputArray].arrInfoSubItems[uiLPClearOutputArray].bIsEnum := FALSE;
																		arrVarInfos[udiCounterClearOutputArray].arrInfoSubItems[uiLPClearOutputArray].sSubItemName := '';
																			arrVarInfos[udiCounterClearOutputArray].arrInfoSubItems[uiLPClearOutputArray].sSubItemType := '';
																				arrVarInfos[udiCounterClearOutputArray].arrInfoSubItems[uiLPClearOutputArray].udiSubItemGroup := 0;
																					arrVarInfos[udiCounterClearOutputArray].arrInfoSubItems[uiLPClearOutputArray].udiSubItemOffset := 0;	
																						arrVarInfos[udiCounterClearOutputArray].arrInfoSubItems[uiLPClearOutputArray].udiSubItemSize := 0;
																							arrVarInfos[udiCounterClearOutputArray].arrInfoSubItems[uiLPClearOutputArray].uiSizeArray := 0;	
																								arrVarInfos[udiCounterClearOutputArray].arrInfoSubItems[uiLPClearOutputArray].sSubItemUnit := '';	
																END_FOR 
			arrAllVarInfosForGV[udiCounterClearOutputArray].sFullSymbolName := '';
				arrAllVarInfosForGV[udiCounterClearOutputArray].sSymbolType := '';	
					arrAllVarInfosForGV[udiCounterClearOutputArray].sSymbolUnit := '';
						arrAllVarInfosForGV[udiCounterClearOutputArray].udiGroup := 0;
							arrAllVarInfosForGV[udiCounterClearOutputArray].udiOffset := 0;	
								arrAllVarInfosForGV[udiCounterClearOutputArray].udiSize := 0;
									arrAllVarInfosForGV[udiCounterClearOutputArray].uiSizeArray := 0;	
		END_IF
		
		FOR byLPClearArraySubItemInfo := 1 TO 12 BY 1 DO
			arrADSInfoSubItem[byLPClearArraySubItemInfo] := 0;
		END_FOR   
		
		//Progress to 1 % when deletign the content of the array
		IF udiCounterClearOutputArray < udiCounterFoundVariablesInt THEN byProgress := 1; END_IF 
		
		IF udiCounterClearOutputArray >= udiCounterFoundVariablesInt THEN 
		
		bErrorIntern := FALSE;
			udiErrorIntern := 0;
				sVarWithError := '';
					udiCounterFoundVariables := 0; 
						udiCounterFoundVariablesInt := 0;
		
		fbADSRead.IDXGRP := ADSIGRP_SYM_UPLOADINFO;
			fbADSRead.IDXOFFS := 0;
				fbADSRead.LEN:= SIZEOF(stSymbolUploadInfo);
					fbADSRead.DESTADDR:= ADR(stSymbolUploadInfo); 
						fbADSRead.READ := TRUE;
		
		IF NOT fbADSRead.BUSY AND NOT fbADSRead.ERR AND byCounterWaitInStep >= rWaitInStep AND stSymbolUploadInfo.udiSymbols > 0 AND uiStateVarToGVInterface = 0 THEN 
			uiStateRead := 2; byCounterWaitInStep := 0; fbADSRead.READ := FALSE; udiCounterSymbol := 1;
		END_IF
			IF timTimout.Q OR FPError.Q OR (byCounterWaitInStep >= rWaitInStep AND stSymbolUploadInfo.udiSymbols <= 0) THEN 
				uiStateRead := 200;
					//Array Error
					IF NOT FPError.Q THEN udiErrorIntern := 1; END_IF	
					//Timout Error
					IF timTimout.Q THEN udiErrorIntern := 2; END_IF		
			END_IF		
				
		byCounterWaitInStep := byCounterWaitInStep + 1;
		
		END_IF	
		
	2: //Read Information about the PLC Variables
		fbADSRead.IDXGRP := ADSIGRP_SYM_UPLOAD;
			fbADSRead.IDXOFFS := udiCounterSymbol;
				fbADSRead.LEN:= SIZEOF(arrSymbols);
					fbADSRead.DESTADDR:= ADR(arrSymbols); 
						fbADSRead.READ := TRUE;
			
		IF NOT fbADSRead.BUSY AND NOT fbADSRead.ERR AND byCounterWaitInStep >= rWaitInStep THEN uiStateRead := 3; byCounterWaitInStep := 0; fbADSRead.READ := FALSE; END_IF
			IF FPError.Q OR timTimout.Q THEN uiStateRead := 200; END_IF	
				//Timout Error	
				IF timTimout.Q THEN udiErrorIntern := 2; END_IF		
					
			IF uiStateRead = 2 THEN byCounterWaitInStep := byCounterWaitInStep + 1; END_IF
				
	3: //Symbol Upload
		MEMCPY(ADR(stADSSymbolUpload),ADR(arrSymbols),SIZEOF(stADSSymbolUpload));
			stADSVarInfo.udiGroup := stADSSymbolUpload.udiGroup;
				stADSVarInfo.udiOffset := stADSSymbolUpload.udiOffset;
					stADSVarInfo.udiSize := stADSSymbolUpload.udiSize;
						stADSVarInfo.udiFlags := stADSSymbolUpload.udiFlags; 
							stADSVarInfo.uiTypeLength := stADSSymbolUpload.uiTypeLength; 
								uiStateRead := 4;
									udiLengthTo_0 := 0;
			//Timout Error					
			IF timTimout.Q THEN uiStateRead := 200; udiErrorIntern := 2; END_IF		
		
	4: //Variable Name and ADS data type
		stADSVarInfo.sAdsDataType := '';
		
		IF stADSSymbolUpload.udiAdsDataType = 33 THEN stADSVarInfo.sAdsDataType := 'ADST_BIT'; END_IF
		IF stADSSymbolUpload.udiAdsDataType = 16 THEN stADSVarInfo.sAdsDataType := 'ADST_INT8'; END_IF 
		IF stADSSymbolUpload.udiAdsDataType = 2 THEN stADSVarInfo.sAdsDataType := 'ADST_INT16'; END_IF
		IF stADSSymbolUpload.udiAdsDataType = 3 THEN stADSVarInfo.sAdsDataType := 'ADST_INT32'; END_IF
		IF stADSSymbolUpload.udiAdsDataType = 20 THEN stADSVarInfo.sAdsDataType := 'ADST_INT64'; END_IF
		IF stADSSymbolUpload.udiAdsDataType = 17 THEN stADSVarInfo.sAdsDataType := 'ADST_UINT8'; END_IF
		IF stADSSymbolUpload.udiAdsDataType = 18 THEN stADSVarInfo.sAdsDataType := 'ADST_UINT16'; END_IF
		IF stADSSymbolUpload.udiAdsDataType = 19 THEN stADSVarInfo.sAdsDataType := 'ADST_UINT32'; END_IF
		IF stADSSymbolUpload.udiAdsDataType = 21 THEN stADSVarInfo.sAdsDataType := 'ADST_UINT64'; END_IF
		IF stADSSymbolUpload.udiAdsDataType = 4 THEN stADSVarInfo.sAdsDataType := 'ADST_REAL32'; END_IF
		IF stADSSymbolUpload.udiAdsDataType = 5 THEN stADSVarInfo.sAdsDataType := 'ADST_REAL64'; END_IF
		IF stADSSymbolUpload.udiAdsDataType = 32 THEN stADSVarInfo.sAdsDataType := 'ADST_REAL80'; END_IF
		IF stADSSymbolUpload.udiAdsDataType = 65 THEN stADSVarInfo.sAdsDataType := 'ADST_BIGTYPE'; END_IF
		IF stADSSymbolUpload.udiAdsDataType = 30 THEN stADSVarInfo.sAdsDataType := 'ADST_STRING'; END_IF
		IF stADSSymbolUpload.udiAdsDataType = 0 THEN stADSVarInfo.sAdsDataType := 'ADST_VOID'; END_IF
		
		stADSVarInfo.sSymbolName := '';
			IF (stADSSymbolUpload.uiNameLength + 30) <= Lynus_Standards.Constants_Communicator.udiArraySizeSymbols THEN  		 
				FOR udiLPSearch_0 := 30 TO (stADSSymbolUpload.uiNameLength + 30) BY 1 DO
					stADSVarInfo.sSymbolName := CONCAT(stADSVarInfo.sSymbolName,F_ToCHR(arrSymbols[udiLPSearch_0]));
						IF arrSymbols[udiLPSearch_0] = 0 THEN udiLengthTo_0 := udiLPSearch_0 - 30; EXIT; END_IF  
				END_FOR 
			END_IF			
				
				IF udiLengthTo_0 <> 0 AND udiLengthTo_0 <= 255 THEN udiFactortLP := (udiLengthTo_0 + 31); udiLengthTo_0 := 0; uiStateRead := 5; END_IF 
					//Timout Error or comment description error
					IF timTimout.Q OR udiLengthTo_0 > 255 THEN 
						IF timTimout.Q THEN uiStateRead := 200; udiErrorIntern := 2; ELSE uiStateRead := 200; udiErrorIntern := 4; END_IF
					END_IF
	
	5: //Symbole Type
		stADSVarInfo.sSymbolType := '';
			IF udiFactortLP < Lynus_Standards.Constants_Communicator.udiArraySizeSymbols THEN
				FOR udiLPSearch_0 := udiFactortLP TO Lynus_Standards.Constants_Communicator.udiArraySizeSymbols BY 1 DO
					stADSVarInfo.sSymbolType := CONCAT(stADSVarInfo.sSymbolType,F_ToCHR(arrSymbols[udiLPSearch_0]));
						IF arrSymbols[udiLPSearch_0] = 0 THEN udiLengthTo_0 := udiLPSearch_0 - udiFactortLP; EXIT; END_IF 
				END_FOR
			END_IF
				
		//Check for mor than 1 Info function ore more than 1 read write function or mor than 1 send/receive function
		IF FIND(stADSVarInfo.sSymbolType,'TSG_Communicator.FB_VarInfo') = 1 THEN byCounterNumberFuctionInfo := byCounterNumberFuctionInfo + 1; END_IF
			IF FIND(stADSVarInfo.sSymbolType,'TSG_Communicator.FB_ReadWrite') = 1 THEN byCounterNumberFuctionReadWrite := byCounterNumberFuctionReadWrite + 1; END_IF
				IF FIND(stADSVarInfo.sSymbolType,'TSG_Communicator.FB_MqttCommunicator') = 1 THEN byCounterSendReceiveFunction := byCounterSendReceiveFunction + 1; END_IF	
			
				IF udiLengthTo_0 <> 0 AND udiLengthTo_0 <= 255 AND udiFactortLP < Lynus_Standards.Constants_Communicator.udiArraySizeSymbols AND byCounterNumberFuctionInfo <= 1 AND byCounterNumberFuctionReadWrite <= 10 AND byCounterSendReceiveFunction <= 1 THEN 
					udiFactortLP := udiFactortLP + udiLengthTo_0 + 1; 
						udiLengthTo_0 := 0; 
							uiStateRead := 6; 
				END_IF 
					IF udiFactortLP >= Lynus_Standards.Constants_Communicator.udiArraySizeSymbols OR timTimout.Q OR udiLengthTo_0 > 255 OR byCounterNumberFuctionInfo > 1 OR byCounterNumberFuctionReadWrite > 10 OR byCounterSendReceiveFunction > 1 THEN
							uiStateRead := 200;
								//Comment lenght Error or timout Error
								IF timTimout.Q THEN udiErrorIntern := 2; END_IF 
								IF udiFactortLP >= Lynus_Standards.Constants_Communicator.udiArraySizeSymbols THEN udiErrorIntern := 3; END_IF 
								IF udiLengthTo_0 > 255 THEN udiErrorIntern := 3; END_IF
								IF byCounterNumberFuctionReadWrite > 10 THEN udiErrorIntern := 7; END_IF 
								IF byCounterNumberFuctionInfo > 1 THEN udiErrorIntern := 8; END_IF 
								IF byCounterSendReceiveFunction > 1 THEN udiErrorIntern := 9; END_IF
					END_IF
					
	6: //Symbol Comment
		stADSVarInfo.sSymbolComment := '';
			IF udiFactortLP < Lynus_Standards.Constants_Communicator.udiArraySizeSymbols THEN
				FOR udiLPSearch_0 := udiFactortLP TO Lynus_Standards.Constants_Communicator.udiArraySizeSymbols BY 1 DO
					stADSVarInfo.sSymbolComment := CONCAT(stADSVarInfo.sSymbolComment,F_ToCHR(arrSymbols[udiLPSearch_0]));
						IF arrSymbols[udiLPSearch_0] = 0 THEN udiLengthTo_0 := udiLPSearch_0 - udiFactortLP; EXIT; END_IF 
				END_FOR
			END_IF
				
				IF udiLengthTo_0 <= 255 AND udiFactortLP < Lynus_Standards.Constants_Communicator.udiArraySizeSymbols THEN udiFactortLP := 0; udiLengthTo_0 := 0; uiStateRead := 7; END_IF 
					IF udiFactortLP >= Lynus_Standards.Constants_Communicator.udiArraySizeSymbols OR timTimout.Q OR udiLengthTo_0 > 255 THEN 
						uiStateRead := 200;
							//Comment lenght Error or timout Error
							IF timTimout.Q THEN udiErrorIntern := 2; END_IF 
							IF udiFactortLP >= Lynus_Standards.Constants_Communicator.udiArraySizeSymbols THEN udiErrorIntern := 3; END_IF 
							IF udiLengthTo_0 > 255 THEN udiErrorIntern := 3; END_IF 
					END_IF
	
	7: //Look it is a variable with the right start information for Lynus
		IF MID(stADSVarInfo.sSymbolComment,14,1) = '{#lynus.ag#()}' THEN 
			IF FIND(stADSVarInfo.sSymbolType,'FB_VarInfo') = 0 AND FIND(stADSVarInfo.sSymbolType,'FB_ReadWrite') = 0 AND FIND(stADSVarInfo.sSymbolType,'FB_MqttCommiunicator') = 0 THEN 
				uiStateRead := 8; 
			ELSE
				uiStateRead := 200;
					udiErrorIntern := 5;
			END_IF 
		ELSE
			uiStateRead := 100; 
		END_IF	
			//Timout Error		
			IF timTimout.Q THEN uiStateRead := 200; udiErrorIntern := 2; END_IF

	8://If it is a array, check the array size and check is standart datatype or not
		//Check Array Size
		IF FIND(stADSVarInfo.sSymbolType,'ARRAY') = 1 THEN 
			//detect array size
			arrFind[1] := FIND(stADSVarInfo.sSymbolType,'[');
				uiValueLower := STRING_TO_UINT(MID(stADSVarInfo.sSymbolType,1,arrFind[1] + 1));
					arrFind[2] := FIND(stADSVarInfo.sSymbolType,']');
			IF arrFind[1] = 7 AND arrFind[2] = 12 THEN
				uiValueHigher := STRING_TO_UINT(MID(stADSVarInfo.sSymbolType,1,arrFind[2] - 1));
			ELSIF arrFind[1] = 7 AND arrFind[2] = 13 THEN
				uiValueHigher := STRING_TO_UINT(MID(stADSVarInfo.sSymbolType,2,arrFind[2] - 2));
			ELSIF arrFind[1] = 7 AND arrFind[2] = 14 THEN
				uiValueHigher := STRING_TO_UINT(MID(stADSVarInfo.sSymbolType,3,arrFind[2] - 3));
			END_IF	
				uiSizeArray := (uiValueHigher - uiValueLower) + 1;
					//Check for 2 or 3 dimensional array
					IF FIND(stADSVarInfo.sSymbolType,',') <> 0 THEN uiSizeArray := Lynus_Standards.Constants_Communicator.bySizeOfValueArray + 1; END_IF
		END_IF
			//Check Datatype
			IF FIND(stADSVarInfo.sSymbolType,'BOOL') = 0 AND FIND(stADSVarInfo.sSymbolType,'BYTE') = 0 AND FIND(stADSVarInfo.sSymbolType,'WORD') = 0 AND FIND(stADSVarInfo.sSymbolType,'DWORD') = 0 AND FIND(stADSVarInfo.sSymbolType,'SINT') = 0 AND
				FIND(stADSVarInfo.sSymbolType,'USINT') = 0 AND FIND(stADSVarInfo.sSymbolType,'INT') = 0 AND FIND(stADSVarInfo.sSymbolType,'UINT') = 0 AND FIND(stADSVarInfo.sSymbolType,'DINT') = 0 AND FIND(stADSVarInfo.sSymbolType,'UDINT') = 0 AND
					FIND(stADSVarInfo.sSymbolType,'LINT') = 0 AND FIND(stADSVarInfo.sSymbolType,'ULINT') = 0 AND FIND(stADSVarInfo.sSymbolType,'LWORD') = 0 AND FIND(stADSVarInfo.sSymbolType,'REAL') = 0 AND FIND(stADSVarInfo.sSymbolType,'LREAL') = 0 AND
						FIND(stADSVarInfo.sSymbolType,'STRING(30)') = 0 AND FIND(stADSVarInfo.sSymbolType,'TIME') = 0 AND FIND(stADSVarInfo.sSymbolType,'TIME_OF_DAY') = 0 AND FIND(stADSVarInfo.sSymbolType,'DATE') = 0 AND FIND(stADSVarInfo.sSymbolType,'DATE_AND_TIME') = 0 AND
			FIND(stADSVarInfo.sSymbolType,'OF BOOL') = 0 AND FIND(stADSVarInfo.sSymbolType,'OF BYTE') = 0 AND FIND(stADSVarInfo.sSymbolType,'OF WORD') = 0 AND FIND(stADSVarInfo.sSymbolType,'OF DWORD') = 0 AND FIND(stADSVarInfo.sSymbolType,'OF SINT') = 0 AND
				FIND(stADSVarInfo.sSymbolType,'OF USINT') = 0 AND FIND(stADSVarInfo.sSymbolType,'OF INT') = 0 AND FIND(stADSVarInfo.sSymbolType,'OF UINT') = 0 AND FIND(stADSVarInfo.sSymbolType,'OF DINT') = 0 AND FIND(stADSVarInfo.sSymbolType,'OF UDINT') = 0 AND
					FIND(stADSVarInfo.sSymbolType,'OF LINT') = 0 AND FIND(stADSVarInfo.sSymbolType,'OF ULINT') = 0 AND FIND(stADSVarInfo.sSymbolType,'OF LWORD') = 0 AND FIND(stADSVarInfo.sSymbolType,'OF REAL') = 0 AND FIND(stADSVarInfo.sSymbolType,'OF LREAL') = 0 AND
						FIND(stADSVarInfo.sSymbolType,'OF STRING(30)') = 0 AND FIND(stADSVarInfo.sSymbolType,'OF TIME') = 0 AND FIND(stADSVarInfo.sSymbolType,'OF TIME_OF_DAY') = 0 AND FIND(stADSVarInfo.sSymbolType,'OF DATE') = 0 AND FIND(stADSVarInfo.sSymbolType,'OF DATE_AND_TIME') = 0 THEN
				bNoStandardDatatypeDetected := TRUE;
			ELSE
				bNoStandardDatatypeDetected := FALSE;
			END_IF	         	   	   				
				//Ckeck String Size
				IF FIND(stADSVarInfo.sSymbolType,'STRING(') <> 0 OR FIND(stADSVarInfo.sSymbolType,'OF STRING(') <> 0 THEN uliSizeOfString := STRING_TO_ULINT(MID(stADSVarInfo.sSymbolType,FIND(stADSVarInfo.sSymbolType,')') - FIND(stADSVarInfo.sSymbolType,'(') - 1,FIND(stADSVarInfo.sSymbolType,'(') + 1)); bStringDetected := TRUE; END_IF 

